LIN {X 0,Y 516.45,Z 515.759,A -85,B 0,C 180,E1 -4943.75,E2 -4943.75} C_VEL
LIN {X 0,Y 516.313,Z 520.47,A -85,B 0,C 180,E1 -4944.924,E2 -4944.924} C_VEL
LIN {X 0,Y 516.373,Z 524.074,A -85,B 0,C 180,E1 -4946.098,E2 -4946.098} C_VEL
LIN {X 0,Y 516.282,Z 525.941,A -85,B 0,C 180,E1 -4946.879,E2 -4946.879} C_VEL
LIN {X 0,Y 516.261,Z 527.348,A -85,B 0,C 180,E1 -4947.659,E2 -4947.659} C_VEL
LIN {X 0,Y 516.16,Z 528.967,A -85,B 0,C 180,E1 -4949.22,E2 -4949.22} C_VEL
LIN {X 0,Y 516.155,Z 529.205,A -85,B 0,C 180,E1 -4950,E2 -4950} C_VEL
LIN {X 0,Y 516.16,Z 529.022,A -85,B 0,C 180,E1 -4950.78,E2 -4950.78} C_VEL
LIN {X 0,Y 516.262,Z 527.473,A -85,B 0,C 180,E1 -4952.341,E2 -4952.341} C_VEL
LIN {X 0,Y 516.283,Z 526.12,A -85,B 0,C 180,E1 -4953.121,E2 -4953.121} C_VEL
LIN {X 0,Y 516.361,Z 523.259,A -85,B 0,C 180,E1 -4954.293,E2 -4954.293} C_VEL
LIN {X 0,Y 516.404,Z 519.379,A -85,B 0,C 180,E1 -4955.467,E2 -4955.467} C_VEL
LIN {X 0,Y 516.485,Z 513.559,A -85,B 0,C 180,E1 -4956.808,E2 -4956.808} C_VEL
LIN {X 0,Y 516.654,Z 506.85,A -85,B 0,C 180,E1 -4958.015,E2 -4958.015} C_VEL
LIN {X 0,Y 516.847,Z 498.704,A -85,B 0,C 180,E1 -4959.194,E2 -4959.194} C_VEL
LIN {X 0,Y 517.103,Z 490.365,A -85,B 0,C 180,E1 -4960.177,E2 -4960.177} C_VEL
LIN {X 0,Y 517.462,Z 480.067,A -85,B 0,C 180,E1 -4961.159,E2 -4961.159} C_VEL
LIN {X 0,Y 517.768,Z 468.543,A -85,B 0,C 180,E1 -4962.039,E2 -4962.039} C_VEL
LIN {X 0,Y 518.054,Z 456.894,A -85,B 0,C 180,E1 -4962.736,E2 -4962.736} C_VEL
LIN {X 0,Y 518.318,Z 444.877,A -85,B 0,C 180,E1 -4963.277,E2 -4963.277} C_VEL
LIN {X 0,Y 518.3,Z 435.908,A -85,B 0,C 180,E1 -4963.59,E2 -4963.59} C_VEL
LIN {X 0,Y 516.365,Z 425.054,A -85,B 0,C 180,E1 -4963.93,E2 -4963.93} C_VEL
LIN {X 0,Y 516.347,Z 420.588,A -85,B 0,C 180,E1 -4966.609,E2 -4966.609} C_VEL
LIN {X 0,Y 516.394,Z 416.475,A -85,B 0,C 180,E1 -4969.065,E2 -4969.065} C_VEL
LIN {X 0,Y 516.487,Z 411.014,A -85,B 0,C 180,E1 -4972.396,E2 -4972.396} C_VEL
LIN {X 0,Y 516.554,Z 406.929,A -85,B 0,C 180,E1 -4974.947,E2 -4974.947} C_VEL
LIN {X 0,Y 516.637,Z 402.398,A -85,B 0,C 180,E1 -4977.844,E2 -4977.844} C_VEL
LIN {X 0,Y 516.679,Z 398.764,A -85,B 0,C 180,E1 -4980.218,E2 -4980.218} C_VEL
LIN {X 0,Y 516.778,Z 394.644,A -85,B 0,C 180,E1 -4982.956,E2 -4982.956} C_VEL
LIN {X 0,Y 516.764,Z 391.166,A -85,B 0,C 180,E1 -4985.313,E2 -4985.313} C_VEL
LIN {X 0,Y 516.883,Z 391.097,A -85,B 0,C 180,E1 -4987.943,E2 -4987.943} C_VEL
LIN {X 0,Y 516.888,Z 391.1,A -85,B 0,C 180,E1 -4990.742,E2 -4990.742} C_VEL
LIN {X 0,Y 516.908,Z 391.096,A -85,B 0,C 180,E1 -4992.829,E2 -4992.829} C_VEL
LIN {X 0,Y 516.885,Z 391.099,A -85,B 0,C 180,E1 -4996.107,E2 -4996.107} C_VEL
LIN {X 0,Y 516.916,Z 391.095,A -85,B 0,C 180,E1 -4998.399,E2 -4998.399} C_VEL
LIN {X 0,Y 516.886,Z 391.097,A -85,B 0,C 180,E1 -5001.284,E2 -5001.284} C_VEL
LIN {X 0,Y 516.874,Z 391.104,A -85,B 0,C 180,E1 -5004.22,E2 -5004.22} C_VEL
LIN {X 0,Y 516.898,Z 391.099,A -85,B 0,C 180,E1 -5007.053,E2 -5007.053} C_VEL
LIN {X 0,Y 516.895,Z 391.098,A -85,B 0,C 180,E1 -5009.796,E2 -5009.796} C_VEL
LIN {X 0,Y 516.932,Z 391.096,A -85,B 0,C 180,E1 -5012.467,E2 -5012.467} C_VEL
LIN {X 0,Y 516.879,Z 391.098,A -85,B 0,C 180,E1 -5015.07,E2 -5015.07} C_VEL
LIN {X 0,Y 516.872,Z 391.102,A -85,B 0,C 180,E1 -5017.622,E2 -5017.622} C_VEL
LIN {X 0,Y 516.936,Z 391.093,A -85,B 0,C 180,E1 -5020.13,E2 -5020.13} C_VEL
LIN {X 0,Y 516.911,Z 391.098,A -85,B 0,C 180,E1 -5022.595,E2 -5022.595} C_VEL
LIN {X 0,Y 516.946,Z 391.092,A -85,B 0,C 180,E1 -5025.03,E2 -5025.03} C_VEL
LIN {X 0,Y 516.969,Z 391.091,A -85,B 0,C 180,E1 -5028.234,E2 -5028.234} C_VEL
LIN {X 0,Y 516.973,Z 391.09,A -85,B 0,C 180,E1 -5031.4,E2 -5031.4} C_VEL
LIN {X 0,Y 517.013,Z 391.083,A -85,B 0,C 180,E1 -5033.757,E2 -5033.757} C_VEL
LIN {X 0,Y 517.085,Z 391.074,A -85,B 0,C 180,E1 -5037.663,E2 -5037.663} C_VEL
LIN {X 0,Y 517.097,Z 391.07,A -85,B 0,C 180,E1 -5040.779,E2 -5040.779} C_VEL
LIN {X 0,Y 517.015,Z 391.083,A -85,B 0,C 180,E1 -5043.117,E2 -5043.117} C_VEL
LIN {X 0,Y 517.013,Z 391.083,A -85,B 0,C 180,E1 -5046.243,E2 -5046.243} C_VEL
LIN {X 0,Y 516.956,Z 391.09,A -85,B 0,C 180,E1 -5049.389,E2 -5049.389} C_VEL
LIN {X 0,Y 516.988,Z 391.089,A -85,B 0,C 180,E1 -5051.824,E2 -5051.824} C_VEL
LIN {X 0,Y 516.948,Z 391.091,A -85,B 0,C 180,E1 -5055.146,E2 -5055.146} C_VEL
LIN {X 0,Y 516.929,Z 391.093,A -85,B 0,C 180,E1 -5058.222,E2 -5058.222} C_VEL
LIN {X 0,Y 516.916,Z 391.098,A -85,B 0,C 180,E1 -5060.701,E2 -5060.701} C_VEL
LIN {X 0,Y 516.894,Z 391.1,A -85,B 0,C 180,E1 -5064.073,E2 -5064.073} C_VEL
LIN {X 0,Y 516.929,Z 391.092,A -85,B 0,C 180,E1 -5066.658,E2 -5066.658} C_VEL
LIN {X 0,Y 516.914,Z 391.096,A -85,B 0,C 180,E1 -5069.524,E2 -5069.524} C_VEL
LIN {X 0,Y 516.899,Z 391.1,A -85,B 0,C 180,E1 -5072.543,E2 -5072.543} C_VEL
LIN {X 0,Y 516.882,Z 391.099,A -85,B 0,C 180,E1 -5075.332,E2 -5075.332} C_VEL
LIN {X 0,Y 516.884,Z 391.101,A -85,B 0,C 180,E1 -5077.943,E2 -5077.943} C_VEL
LIN {X 0,Y 516.888,Z 391.099,A -85,B 0,C 180,E1 -5080.741,E2 -5080.741} C_VEL
LIN {X 0,Y 516.887,Z 391.103,A -85,B 0,C 180,E1 -5082.831,E2 -5082.831} C_VEL
LIN {X 0,Y 516.926,Z 391.094,A -85,B 0,C 180,E1 -5085.01,E2 -5085.01} C_VEL
LIN {X 0,Y 516.919,Z 391.097,A -85,B 0,C 180,E1 -5088.398,E2 -5088.398} C_VEL
LIN {X 0,Y 516.884,Z 391.104,A -85,B 0,C 180,E1 -5091.284,E2 -5091.284} C_VEL
LIN {X 0,Y 516.901,Z 391.162,A -85,B 0,C 180,E1 -5092.4,E2 -5092.4} C_VEL
LIN {X 0,Y 517.556,Z 395.906,A -85,B 0,C 180,E1 -5094.563,E2 -5094.563} C_VEL
LIN {X 0,Y 517.418,Z 402.548,A -85,B 0,C 180,E1 -5097.367,E2 -5097.367} C_VEL
LIN {X 0,Y 517.231,Z 410.058,A -85,B 0,C 180,E1 -5100.414,E2 -5100.414} C_VEL
LIN {X 0,Y 517.02,Z 417.541,A -85,B 0,C 180,E1 -5103.347,E2 -5103.347} C_VEL
LIN {X 0,Y 516.858,Z 425.407,A -85,B 0,C 180,E1 -5106.351,E2 -5106.351} C_VEL
LIN {X 0,Y 516.751,Z 433.272,A -85,B 0,C 180,E1 -5109.292,E2 -5109.292} C_VEL
LIN {X 0,Y 516.585,Z 441.385,A -85,B 0,C 180,E1 -5112.238,E2 -5112.238} C_VEL
LIN {X 0,Y 516.514,Z 449.143,A -85,B 0,C 180,E1 -5115.032,E2 -5115.032} C_VEL
LIN {X 0,Y 516.487,Z 452.291,A -85,B 0,C 180,E1 -5116.111,E2 -5116.111} C_VEL
LIN {X 0,Y 518.462,Z 464.61,A -85,B 0,C 180,E1 -5116.452,E2 -5116.452} C_VEL
LIN {X 0,Y 518.211,Z 477.648,A -85,B 0,C 180,E1 -5116.92,E2 -5116.92} C_VEL
LIN {X 0,Y 517.922,Z 490.006,A -85,B 0,C 180,E1 -5117.532,E2 -5117.532} C_VEL
LIN {X 0,Y 517.653,Z 501.19,A -85,B 0,C 180,E1 -5118.249,E2 -5118.249} C_VEL
LIN {X 0,Y 517.34,Z 512.104,A -85,B 0,C 180,E1 -5119.135,E2 -5119.135} C_VEL
LIN {X 0,Y 517.031,Z 521.003,A -85,B 0,C 180,E1 -5120.02,E2 -5120.02} C_VEL
LIN {X 0,Y 516.773,Z 530.675,A -85,B 0,C 180,E1 -5121.199,E2 -5121.199} C_VEL
LIN {X 0,Y 516.563,Z 538.374,A -85,B 0,C 180,E1 -5122.377,E2 -5122.377} C_VEL
LIN {X 0,Y 516.427,Z 545.472,A -85,B 0,C 180,E1 -5123.75,E2 -5123.75} C_VEL
LIN {X 0,Y 516.313,Z 550.193,A -85,B 0,C 180,E1 -5124.924,E2 -5124.924} C_VEL
LIN {X 0,Y 516.354,Z 553.803,A -85,B 0,C 180,E1 -5126.098,E2 -5126.098} C_VEL
LIN {X 0,Y 516.282,Z 555.663,A -85,B 0,C 180,E1 -5126.879,E2 -5126.879} C_VEL
LIN {X 0,Y 516.261,Z 557.058,A -85,B 0,C 180,E1 -5127.659,E2 -5127.659} C_VEL
LIN {X 0,Y 516.16,Z 558.659,A -85,B 0,C 180,E1 -5129.22,E2 -5129.22} C_VEL
LIN {X 0,Y 516.154,Z 558.875,A -85,B 0,C 180,E1 -5130,E2 -5130} C_VEL
LIN {X 0,Y 516.192,Z 558.054,A -85,B 0,C 180,E1 -5131.56,E2 -5131.56} C_VEL
LIN {X 0,Y 516.261,Z 557.061,A -85,B 0,C 180,E1 -5132.341,E2 -5132.341} C_VEL
LIN {X 0,Y 516.282,Z 555.667,A -85,B 0,C 180,E1 -5133.121,E2 -5133.121} C_VEL
LIN {X 0,Y 516.326,Z 552.733,A -85,B 0,C 180,E1 -5134.293,E2 -5134.293} C_VEL
LIN {X 0,Y 516.383,Z 548.761,A -85,B 0,C 180,E1 -5135.467,E2 -5135.467} C_VEL
LIN {X 0,Y 516.465,Z 543.473,A -85,B 0,C 180,E1 -5136.679,E2 -5136.679} C_VEL
LIN {X 0,Y 516.597,Z 537.214,A -85,B 0,C 180,E1 -5137.819,E2 -5137.819} C_VEL
LIN {X 0,Y 516.807,Z 529.186,A -85,B 0,C 180,E1 -5138.997,E2 -5138.997} C_VEL
LIN {X 0,Y 517.031,Z 521.005,A -85,B 0,C 180,E1 -5139.98,E2 -5139.98} C_VEL
LIN {X 0,Y 517.382,Z 511.032,A -85,B 0,C 180,E1 -5140.963,E2 -5140.963} C_VEL
LIN {X 0,Y 517.647,Z 501.194,A -85,B 0,C 180,E1 -5141.751,E2 -5141.751} C_VEL
LIN {X 0,Y 517.933,Z 490.041,A -85,B 0,C 180,E1 -5142.466,E2 -5142.466} C_VEL
LIN {X 0,Y 518.191,Z 477.642,A -85,B 0,C 180,E1 -5143.081,E2 -5143.081} C_VEL
LIN {X 0,Y 518.495,Z 464.607,A -85,B 0,C 180,E1 -5143.547,E2 -5143.547} C_VEL
LIN {X 0,Y 516.475,Z 452.075,A -85,B 0,C 180,E1 -5143.902,E2 -5143.902} C_VEL
LIN {X 0,Y 516.54,Z 444.494,A -85,B 0,C 180,E1 -5146.602,E2 -5146.602} C_VEL
LIN {X 0,Y 516.686,Z 436.567,A -85,B 0,C 180,E1 -5149.466,E2 -5149.466} C_VEL
LIN {X 0,Y 516.797,Z 428.777,A -85,B 0,C 180,E1 -5152.382,E2 -5152.382} C_VEL
LIN {X 0,Y 516.958,Z 420.911,A -85,B 0,C 180,E1 -5155.356,E2 -5155.356} C_VEL
LIN {X 0,Y 517.163,Z 413.048,A -85,B 0,C 180,E1 -5158.401,E2 -5158.401} C_VEL
LIN {X 0,Y 517.356,Z 405.213,A -85,B 0,C 180,E1 -5161.533,E2 -5161.533} C_VEL
LIN {X 0,Y 517.492,Z 399.121,A -85,B 0,C 180,E1 -5164.062,E2 -5164.062} C_VEL
LIN {X 0,Y 517.531,Z 395.238,A -85,B 0,C 180,E1 -5165.728,E2 -5165.728} C_VEL
LIN {X 0,Y 516.884,Z 391.103,A -85,B 0,C 180,E1 -5167.662,E2 -5167.662} C_VEL
LIN {X 0,Y 516.886,Z 391.1,A -85,B 0,C 180,E1 -5170.741,E2 -5170.741} C_VEL
LIN {X 0,Y 516.907,Z 391.096,A -85,B 0,C 180,E1 -5172.829,E2 -5172.829} C_VEL
LIN {X 0,Y 516.925,Z 391.095,A -85,B 0,C 180,E1 -5175.01,E2 -5175.01} C_VEL
LIN {X 0,Y 516.917,Z 391.094,A -85,B 0,C 180,E1 -5178.398,E2 -5178.398} C_VEL
LIN {X 0,Y 516.884,Z 391.098,A -85,B 0,C 180,E1 -5181.284,E2 -5181.284} C_VEL
LIN {X 0,Y 516.891,Z 391.101,A -85,B 0,C 180,E1 -5184.221,E2 -5184.221} C_VEL
LIN {X 0,Y 516.897,Z 391.099,A -85,B 0,C 180,E1 -5187.053,E2 -5187.053} C_VEL
LIN {X 0,Y 516.894,Z 391.096,A -85,B 0,C 180,E1 -5189.796,E2 -5189.796} C_VEL
LIN {X 0,Y 516.93,Z 391.096,A -85,B 0,C 180,E1 -5192.467,E2 -5192.467} C_VEL
LIN {X 0,Y 516.877,Z 391.099,A -85,B 0,C 180,E1 -5195.07,E2 -5195.07} C_VEL
LIN {X 0,Y 516.87,Z 391.103,A -85,B 0,C 180,E1 -5197.622,E2 -5197.622} C_VEL
LIN {X 0,Y 516.935,Z 391.092,A -85,B 0,C 180,E1 -5200.13,E2 -5200.13} C_VEL
LIN {X 0,Y 516.932,Z 391.095,A -85,B 0,C 180,E1 -5202.596,E2 -5202.596} C_VEL
LIN {X 0,Y 516.945,Z 391.091,A -85,B 0,C 180,E1 -5205.03,E2 -5205.03} C_VEL
LIN {X 0,Y 517.007,Z 391.087,A -85,B 0,C 180,E1 -5208.235,E2 -5208.235} C_VEL
LIN {X 0,Y 516.972,Z 391.09,A -85,B 0,C 180,E1 -5211.4,E2 -5211.4} C_VEL
LIN {X 0,Y 517.012,Z 391.083,A -85,B 0,C 180,E1 -5213.757,E2 -5213.757} C_VEL
LIN {X 0,Y 517.085,Z 391.072,A -85,B 0,C 180,E1 -5217.663,E2 -5217.663} C_VEL
LIN {X 0,Y 517.096,Z 391.071,A -85,B 0,C 180,E1 -5220.779,E2 -5220.779} C_VEL
LIN {X 0,Y 517.014,Z 391.085,A -85,B 0,C 180,E1 -5223.117,E2 -5223.117} C_VEL
LIN {X 0,Y 517.012,Z 391.083,A -85,B 0,C 180,E1 -5226.243,E2 -5226.243} C_VEL
LIN {X 0,Y 516.956,Z 391.089,A -85,B 0,C 180,E1 -5229.389,E2 -5229.389} C_VEL
LIN {X 0,Y 516.986,Z 391.089,A -85,B 0,C 180,E1 -5231.824,E2 -5231.824} C_VEL
LIN {X 0,Y 516.947,Z 391.092,A -85,B 0,C 180,E1 -5235.147,E2 -5235.147} C_VEL
LIN {X 0,Y 516.919,Z 391.095,A -85,B 0,C 180,E1 -5238.223,E2 -5238.223} C_VEL
LIN {X 0,Y 516.915,Z 391.097,A -85,B 0,C 180,E1 -5240.701,E2 -5240.701} C_VEL
LIN {X 0,Y 516.893,Z 391.101,A -85,B 0,C 180,E1 -5244.073,E2 -5244.073} C_VEL
LIN {X 0,Y 516.928,Z 391.091,A -85,B 0,C 180,E1 -5246.658,E2 -5246.658} C_VEL
LIN {X 0,Y 516.913,Z 391.097,A -85,B 0,C 180,E1 -5249.524,E2 -5249.524} C_VEL
LIN {X 0,Y 516.898,Z 391.1,A -85,B 0,C 180,E1 -5252.543,E2 -5252.543} C_VEL
LIN {X 0,Y 516.886,Z 391.098,A -85,B 0,C 180,E1 -5255.333,E2 -5255.333} C_VEL
LIN {X 0,Y 516.884,Z 391.1,A -85,B 0,C 180,E1 -5257.943,E2 -5257.943} C_VEL
LIN {X 0,Y 516.887,Z 391.098,A -85,B 0,C 180,E1 -5260.742,E2 -5260.742} C_VEL
LIN {X 0,Y 516.885,Z 391.102,A -85,B 0,C 180,E1 -5262.832,E2 -5262.832} C_VEL
LIN {X 0,Y 516.925,Z 391.095,A -85,B 0,C 180,E1 -5265.01,E2 -5265.01} C_VEL
LIN {X 0,Y 516.918,Z 391.096,A -85,B 0,C 180,E1 -5268.399,E2 -5268.399} C_VEL
LIN {X 0,Y 516.884,Z 391.098,A -85,B 0,C 180,E1 -5270.301,E2 -5270.301} C_VEL
LIN {X 0,Y 516.213,Z 391.184,A -85,B 0,C 180,E1 -5270.951,E2 -5270.951} C_VEL
LIN {X 0,Y 513.364,Z 391.538,A -85,B 0,C 180,E1 -5272.007,E2 -5272.007} C_VEL
LIN {X 0,Y 510.941,Z 391.842,A -85,B 0,C 180,E1 -5272.857,E2 -5272.857} C_VEL
LIN {X 0,Y 509.874,Z 391.975,A -85,B 0,C 180,E1 -5273.513,E2 -5273.513} C_VEL
LIN {X 0,Y 509.774,Z 391.985,A -85,B 0,C 180,E1 -5273.736,E2 -5273.736} C_VEL
LIN {X 0,Y 509.742,Z 391.992,A -85,B 0,C 180,E1 -5274.615,E2 -5274.615} C_VEL
LIN {X 0,Y 509.714,Z 395.641,A -85,B 0,C 180,E1 -5277.254,E2 -5277.254} C_VEL
LIN {X 0,Y 509.61,Z 400.227,A -85,B 0,C 180,E1 -5280.323,E2 -5280.323} C_VEL
LIN {X 0,Y 509.541,Z 404.185,A -85,B 0,C 180,E1 -5282.925,E2 -5282.925} C_VEL
LIN {X 0,Y 509.502,Z 408.276,A -85,B 0,C 180,E1 -5285.561,E2 -5285.561} C_VEL
LIN {X 0,Y 509.373,Z 412.339,A -85,B 0,C 180,E1 -5288.128,E2 -5288.128} C_VEL
LIN {X 0,Y 509.324,Z 416.434,A -85,B 0,C 180,E1 -5290.66,E2 -5290.66} C_VEL
LIN {X 0,Y 509.306,Z 420.558,A -85,B 0,C 180,E1 -5293.155,E2 -5293.155} C_VEL
LIN {X 0,Y 509.279,Z 425.464,A -85,B 0,C 180,E1 -5295.987,E2 -5295.987} C_VEL
LIN {X 0,Y 511.505,Z 437.605,A -85,B 0,C 180,E1 -5296.366,E2 -5296.366} C_VEL
LIN {X 0,Y 511.345,Z 450.083,A -85,B 0,C 180,E1 -5296.842,E2 -5296.842} C_VEL
LIN {X 0,Y 511.029,Z 462.423,A -85,B 0,C 180,E1 -5297.48,E2 -5297.48} C_VEL
LIN {X 0,Y 510.715,Z 474.284,A -85,B 0,C 180,E1 -5298.289,E2 -5298.289} C_VEL
LIN {X 0,Y 510.319,Z 484.759,A -85,B 0,C 180,E1 -5299.185,E2 -5299.185} C_VEL
LIN {X 0,Y 510.061,Z 493.315,A -85,B 0,C 180,E1 -5300.082,E2 -5300.082} C_VEL
LIN {X 0,Y 509.82,Z 501.194,A -85,B 0,C 180,E1 -5301.078,E2 -5301.078} C_VEL
LIN {X 0,Y 509.56,Z 508.9,A -85,B 0,C 180,E1 -5302.272,E2 -5302.272} C_VEL
LIN {X 0,Y 509.387,Z 515.966,A -85,B 0,C 180,E1 -5303.663,E2 -5303.663} C_VEL
LIN {X 0,Y 509.248,Z 520.676,A -85,B 0,C 180,E1 -5304.853,E2 -5304.853} C_VEL
LIN {X 0,Y 509.303,Z 524.279,A -85,B 0,C 180,E1 -5306.044,E2 -5306.044} C_VEL
LIN {X 0,Y 509.201,Z 526.146,A -85,B 0,C 180,E1 -5306.835,E2 -5306.835} C_VEL
LIN {X 0,Y 509.19,Z 527.552,A -85,B 0,C 180,E1 -5307.627,E2 -5307.627} C_VEL
LIN {X 0,Y 509.074,Z 529.171,A -85,B 0,C 180,E1 -5309.209,E2 -5309.209} C_VEL
LIN {X 0,Y 509.066,Z 529.408,A -85,B 0,C 180,E1 -5310,E2 -5310} C_VEL
LIN {X 0,Y 509.074,Z 529.225,A -85,B 0,C 180,E1 -5310.791,E2 -5310.791} C_VEL
LIN {X 0,Y 509.19,Z 527.676,A -85,B 0,C 180,E1 -5312.373,E2 -5312.373} C_VEL
LIN {X 0,Y 509.202,Z 526.323,A -85,B 0,C 180,E1 -5313.165,E2 -5313.165} C_VEL
LIN {X 0,Y 509.282,Z 523.461,A -85,B 0,C 180,E1 -5314.353,E2 -5314.353} C_VEL
LIN {X 0,Y 509.346,Z 519.581,A -85,B 0,C 180,E1 -5315.543,E2 -5315.543} C_VEL
LIN {X 0,Y 509.412,Z 514.576,A -85,B 0,C 180,E1 -5316.734,E2 -5316.734} C_VEL
LIN {X 0,Y 509.597,Z 508.273,A -85,B 0,C 180,E1 -5317.927,E2 -5317.927} C_VEL
LIN {X 0,Y 509.777,Z 500.383,A -85,B 0,C 180,E1 -5319.122,E2 -5319.122} C_VEL
LIN {X 0,Y 510.085,Z 492.336,A -85,B 0,C 180,E1 -5320.118,E2 -5320.118} C_VEL
LIN {X 0,Y 510.414,Z 482.517,A -85,B 0,C 180,E1 -5321.115,E2 -5321.115} C_VEL
LIN {X 0,Y 510.706,Z 472.858,A -85,B 0,C 180,E1 -5321.913,E2 -5321.913} C_VEL
LIN {X 0,Y 511.034,Z 461.886,A -85,B 0,C 180,E1 -5322.641,E2 -5322.641} C_VEL
LIN {X 0,Y 511.332,Z 449.841,A -85,B 0,C 180,E1 -5323.26,E2 -5323.26} C_VEL
LIN {X 0,Y 511.473,Z 437.271,A -85,B 0,C 180,E1 -5323.737,E2 -5323.737} C_VEL
LIN {X 0,Y 509.275,Z 425.263,A -85,B 0,C 180,E1 -5324.128,E2 -5324.128} C_VEL
LIN {X 0,Y 509.288,Z 420.721,A -85,B 0,C 180,E1 -5326.846,E2 -5326.846} C_VEL
LIN {X 0,Y 509.318,Z 416.596,A -85,B 0,C 180,E1 -5329.34,E2 -5329.34} C_VEL
LIN {X 0,Y 509.425,Z 411.586,A -85,B 0,C 180,E1 -5332.432,E2 -5332.432} C_VEL
LIN {X 0,Y 509.493,Z 407.051,A -85,B 0,C 180,E1 -5335.317,E2 -5335.317} C_VEL
LIN {X 0,Y 509.572,Z 402.861,A -85,B 0,C 180,E1 -5338.031,E2 -5338.031} C_VEL
LIN {X 0,Y 509.653,Z 398.017,A -85,B 0,C 180,E1 -5341.244,E2 -5341.244} C_VEL
LIN {X 0,Y 509.748,Z 394.722,A -85,B 0,C 180,E1 -5343.469,E2 -5343.469} C_VEL
LIN {X 0,Y 509.738,Z 391.993,A -85,B 0,C 180,E1 -5345.386,E2 -5345.386} C_VEL
LIN {X 0,Y 509.853,Z 391.976,A -85,B 0,C 180,E1 -5348.338,E2 -5348.338} C_VEL
LIN {X 0,Y 509.861,Z 391.974,A -85,B 0,C 180,E1 -5351.425,E2 -5351.425} C_VEL
LIN {X 0,Y 509.842,Z 391.976,A -85,B 0,C 180,E1 -5354.67,E2 -5354.67} C_VEL
LIN {X 0,Y 509.859,Z 391.973,A -85,B 0,C 180,E1 -5358.103,E2 -5358.103} C_VEL
LIN {X 0,Y 509.851,Z 391.98,A -85,B 0,C 180,E1 -5360.648,E2 -5360.648} C_VEL
LIN {X 0,Y 509.828,Z 391.978,A -85,B 0,C 180,E1 -5363.647,E2 -5363.647} C_VEL
LIN {X 0,Y 509.862,Z 391.974,A -85,B 0,C 180,E1 -5366.539,E2 -5366.539} C_VEL
LIN {X 0,Y 509.849,Z 391.977,A -85,B 0,C 180,E1 -5369.334,E2 -5369.334} C_VEL
LIN {X 0,Y 509.897,Z 391.969,A -85,B 0,C 180,E1 -5372.055,E2 -5372.055} C_VEL
LIN {X 0,Y 509.844,Z 391.976,A -85,B 0,C 180,E1 -5374.702,E2 -5374.702} C_VEL
LIN {X 0,Y 509.83,Z 391.979,A -85,B 0,C 180,E1 -5377.458,E2 -5377.458} C_VEL
LIN {X 0,Y 509.921,Z 391.969,A -85,B 0,C 180,E1 -5379.845,E2 -5379.845} C_VEL
LIN {X 0,Y 509.878,Z 391.973,A -85,B 0,C 180,E1 -5383.174,E2 -5383.174} C_VEL
LIN {X 0,Y 509.868,Z 391.972,A -85,B 0,C 180,E1 -5385.634,E2 -5385.634} C_VEL
LIN {X 0,Y 509.916,Z 391.965,A -85,B 0,C 180,E1 -5388.875,E2 -5388.875} C_VEL
LIN {X 0,Y 509.956,Z 391.962,A -85,B 0,C 180,E1 -5392.078,E2 -5392.078} C_VEL
LIN {X 0,Y 509.985,Z 391.96,A -85,B 0,C 180,E1 -5394.464,E2 -5394.464} C_VEL
LIN {X 0,Y 510.056,Z 391.949,A -85,B 0,C 180,E1 -5397.631,E2 -5397.631} C_VEL
LIN {X 0,Y 510.067,Z 391.946,A -85,B 0,C 180,E1 -5400.789,E2 -5400.789} C_VEL
LIN {X 0,Y 509.957,Z 391.962,A -85,B 0,C 180,E1 -5403.16,E2 -5403.16} C_VEL
LIN {X 0,Y 509.981,Z 391.959,A -85,B 0,C 180,E1 -5406.33,E2 -5406.33} C_VEL
LIN {X 0,Y 509.92,Z 391.969,A -85,B 0,C 180,E1 -5408.72,E2 -5408.72} C_VEL
LIN {X 0,Y 509.955,Z 391.966,A -85,B 0,C 180,E1 -5411.93,E2 -5411.93} C_VEL
LIN {X 0,Y 509.897,Z 391.971,A -85,B 0,C 180,E1 -5415.242,E2 -5415.242} C_VEL
LIN {X 0,Y 509.892,Z 391.969,A -85,B 0,C 180,E1 -5418.001,E2 -5418.001} C_VEL
LIN {X 0,Y 509.854,Z 391.976,A -85,B 0,C 180,E1 -5421.002,E2 -5421.002} C_VEL
LIN {X 0,Y 509.826,Z 391.98,A -85,B 0,C 180,E1 -5423.564,E2 -5423.564} C_VEL
LIN {X 0,Y 509.915,Z 391.966,A -85,B 0,C 180,E1 -5426.379,E2 -5426.379} C_VEL
LIN {X 0,Y 509.88,Z 391.972,A -85,B 0,C 180,E1 -5428.844,E2 -5428.844} C_VEL
LIN {X 0,Y 509.823,Z 391.978,A -85,B 0,C 180,E1 -5431.59,E2 -5431.59} C_VEL
LIN {X 0,Y 509.855,Z 391.977,A -85,B 0,C 180,E1 -5434.413,E2 -5434.413} C_VEL
LIN {X 0,Y 509.822,Z 391.981,A -85,B 0,C 180,E1 -5437.341,E2 -5437.341} C_VEL
LIN {X 0,Y 509.841,Z 391.975,A -85,B 0,C 180,E1 -5440.382,E2 -5440.382} C_VEL
LIN {X 0,Y 509.827,Z 391.98,A -85,B 0,C 180,E1 -5443.062,E2 -5443.062} C_VEL
LIN {X 0,Y 509.834,Z 391.978,A -85,B 0,C 180,E1 -5445.792,E2 -5445.792} C_VEL
LIN {X 0,Y 509.86,Z 391.976,A -85,B 0,C 180,E1 -5448.575,E2 -5448.575} C_VEL
LIN {X 0,Y 509.857,Z 391.977,A -85,B 0,C 180,E1 -5451.786,E2 -5451.786} C_VEL
LIN {X 0,Y 509.885,Z 392.202,A -85,B 0,C 180,E1 -5452.291,E2 -5452.291} C_VEL
LIN {X 0,Y 510.552,Z 396.544,A -85,B 0,C 180,E1 -5454.308,E2 -5454.308} C_VEL
LIN {X 0,Y 510.418,Z 403.106,A -85,B 0,C 180,E1 -5457.131,E2 -5457.131} C_VEL
LIN {X 0,Y 510.25,Z 409.598,A -85,B 0,C 180,E1 -5459.819,E2 -5459.819} C_VEL
LIN {X 0,Y 509.982,Z 417.433,A -85,B 0,C 180,E1 -5462.95,E2 -5462.95} C_VEL
LIN {X 0,Y 509.839,Z 424.175,A -85,B 0,C 180,E1 -5465.572,E2 -5465.572} C_VEL
LIN {X 0,Y 509.7,Z 432.031,A -85,B 0,C 180,E1 -5468.568,E2 -5468.568} C_VEL
LIN {X 0,Y 509.573,Z 439.949,A -85,B 0,C 180,E1 -5471.505,E2 -5471.505} C_VEL
LIN {X 0,Y 509.445,Z 449.296,A -85,B 0,C 180,E1 -5474.946,E2 -5474.946} C_VEL
LIN {X 0,Y 509.401,Z 452.081,A -85,B 0,C 180,E1 -5475.914,E2 -5475.914} C_VEL
LIN {X 0,Y 511.546,Z 465.241,A -85,B 0,C 180,E1 -5476.291,E2 -5476.291} C_VEL
LIN {X 0,Y 511.259,Z 478.575,A -85,B 0,C 180,E1 -5476.789,E2 -5476.789} C_VEL
LIN {X 0,Y 510.946,Z 491.12,A -85,B 0,C 180,E1 -5477.434,E2 -5477.434} C_VEL
LIN {X 0,Y 510.618,Z 502.299,A -85,B 0,C 180,E1 -5478.186,E2 -5478.186} C_VEL
LIN {X 0,Y 510.309,Z 512.972,A -85,B 0,C 180,E1 -5479.084,E2 -5479.084} C_VEL
LIN {X 0,Y 509.954,Z 522.587,A -85,B 0,C 180,E1 -5480.08,E2 -5480.08} C_VEL
LIN {X 0,Y 509.711,Z 530.47,A -85,B 0,C 180,E1 -5481.076,E2 -5481.076} C_VEL
LIN {X 0,Y 509.513,Z 538.17,A -85,B 0,C 180,E1 -5482.271,E2 -5482.271} C_VEL
LIN {X 0,Y 509.328,Z 545.267,A -85,B 0,C 180,E1 -5483.662,E2 -5483.662} C_VEL
LIN {X 0,Y 509.245,Z 549.989,A -85,B 0,C 180,E1 -5484.853,E2 -5484.853} C_VEL
LIN {X 0,Y 509.25,Z 553.599,A -85,B 0,C 180,E1 -5486.043,E2 -5486.043} C_VEL
LIN {X 0,Y 509.2,Z 555.459,A -85,B 0,C 180,E1 -5486.835,E2 -5486.835} C_VEL
LIN {X 0,Y 509.19,Z 556.854,A -85,B 0,C 180,E1 -5487.627,E2 -5487.627} C_VEL
LIN {X 0,Y 509.073,Z 558.455,A -85,B 0,C 180,E1 -5489.209,E2 -5489.209} C_VEL
LIN {X 0,Y 509.065,Z 558.671,A -85,B 0,C 180,E1 -5490,E2 -5490} C_VEL
LIN {X 0,Y 509.113,Z 557.85,A -85,B 0,C 180,E1 -5491.582,E2 -5491.582} C_VEL
LIN {X 0,Y 509.19,Z 556.858,A -85,B 0,C 180,E1 -5492.373,E2 -5492.373} C_VEL
LIN {X 0,Y 509.2,Z 555.463,A -85,B 0,C 180,E1 -5493.165,E2 -5493.165} C_VEL
LIN {X 0,Y 509.216,Z 552.528,A -85,B 0,C 180,E1 -5494.353,E2 -5494.353} C_VEL
LIN {X 0,Y 509.305,Z 548.557,A -85,B 0,C 180,E1 -5495.543,E2 -5495.543} C_VEL
LIN {X 0,Y 509.402,Z 542.902,A -85,B 0,C 180,E1 -5496.844,E2 -5496.844} C_VEL
LIN {X 0,Y 509.573,Z 535.772,A -85,B 0,C 180,E1 -5498.127,E2 -5498.127} C_VEL
LIN {X 0,Y 509.793,Z 527.489,A -85,B 0,C 180,E1 -5499.322,E2 -5499.322} C_VEL
LIN {X 0,Y 510.055,Z 519,A -85,B 0,C 180,E1 -5500.319,E2 -5500.319} C_VEL
LIN {X 0,Y 510.423,Z 508.512,A -85,B 0,C 180,E1 -5501.315,E2 -5501.315} C_VEL
LIN {X 0,Y 510.696,Z 497.21,A -85,B 0,C 180,E1 -5502.179,E2 -5502.179} C_VEL
LIN {X 0,Y 511.071,Z 486.762,A -85,B 0,C 180,E1 -5502.811,E2 -5502.811} C_VEL
LIN {X 0,Y 511.313,Z 475.096,A -85,B 0,C 180,E1 -5503.361,E2 -5503.361} C_VEL
LIN {X 0,Y 511.434,Z 464.398,A -85,B 0,C 180,E1 -5503.737,E2 -5503.737} C_VEL
LIN {X 0,Y 509.387,Z 451.894,A -85,B 0,C 180,E1 -5504.099,E2 -5504.099} C_VEL
LIN {X 0,Y 509.468,Z 444.335,A -85,B 0,C 180,E1 -5506.839,E2 -5506.839} C_VEL
LIN {X 0,Y 509.627,Z 436.478,A -85,B 0,C 180,E1 -5509.747,E2 -5509.747} C_VEL
LIN {X 0,Y 509.753,Z 429.156,A -85,B 0,C 180,E1 -5512.521,E2 -5512.521} C_VEL
LIN {X 0,Y 509.942,Z 420.8,A -85,B 0,C 180,E1 -5515.73,E2 -5515.73} C_VEL
LIN {X 0,Y 510.14,Z 412.946,A -85,B 0,C 180,E1 -5518.828,E2 -5518.828} C_VEL
LIN {X 0,Y 510.352,Z 405.128,A -85,B 0,C 180,E1 -5522.018,E2 -5522.018} C_VEL
LIN {X 0,Y 510.568,Z 398.479,A -85,B 0,C 180,E1 -5524.837,E2 -5524.837} C_VEL
LIN {X 0,Y 510.38,Z 395.183,A -85,B 0,C 180,E1 -5526.307,E2 -5526.307} C_VEL
LIN {X 0,Y 509.847,Z 391.98,A -85,B 0,C 180,E1 -5527.837,E2 -5527.837} C_VEL
LIN {X 0,Y 509.841,Z 391.978,A -85,B 0,C 180,E1 -5530.698,E2 -5530.698} C_VEL
LIN {X 0,Y 509.829,Z 391.982,A -85,B 0,C 180,E1 -5533.571,E2 -5533.571} C_VEL
LIN {X 0,Y 509.82,Z 391.977,A -85,B 0,C 180,E1 -5536.428,E2 -5536.428} C_VEL
LIN {X 0,Y 509.841,Z 391.976,A -85,B 0,C 180,E1 -5539.302,E2 -5539.302} C_VEL
LIN {X 0,Y 509.854,Z 391.975,A -85,B 0,C 180,E1 -5541.786,E2 -5541.786} C_VEL
LIN {X 0,Y 509.846,Z 391.976,A -85,B 0,C 180,E1 -5544.623,E2 -5544.623} C_VEL
LIN {X 0,Y 509.863,Z 391.976,A -85,B 0,C 180,E1 -5547.481,E2 -5547.481} C_VEL
LIN {X 0,Y 509.86,Z 391.973,A -85,B 0,C 180,E1 -5550.274,E2 -5550.274} C_VEL
LIN {X 0,Y 509.887,Z 391.971,A -85,B 0,C 180,E1 -5552.944,E2 -5552.944} C_VEL
LIN {X 0,Y 509.853,Z 391.976,A -85,B 0,C 180,E1 -5555.573,E2 -5555.573} C_VEL
LIN {X 0,Y 509.824,Z 391.98,A -85,B 0,C 180,E1 -5558.149,E2 -5558.149} C_VEL
LIN {X 0,Y 509.867,Z 391.974,A -85,B 0,C 180,E1 -5560.682,E2 -5560.682} C_VEL
LIN {X 0,Y 509.887,Z 391.971,A -85,B 0,C 180,E1 -5563.175,E2 -5563.175} C_VEL
LIN {X 0,Y 509.867,Z 391.971,A -85,B 0,C 180,E1 -5565.634,E2 -5565.634} C_VEL
LIN {X 0,Y 509.924,Z 391.965,A -85,B 0,C 180,E1 -5568.875,E2 -5568.875} C_VEL
LIN {X 0,Y 509.954,Z 391.962,A -85,B 0,C 180,E1 -5572.079,E2 -5572.079} C_VEL
LIN {X 0,Y 509.984,Z 391.96,A -85,B 0,C 180,E1 -5574.464,E2 -5574.464} C_VEL
LIN {X 0,Y 510.056,Z 391.948,A -85,B 0,C 180,E1 -5577.631,E2 -5577.631} C_VEL
LIN {X 0,Y 510.066,Z 391.947,A -85,B 0,C 180,E1 -5580.79,E2 -5580.79} C_VEL
LIN {X 0,Y 509.956,Z 391.964,A -85,B 0,C 180,E1 -5583.16,E2 -5583.16} C_VEL
LIN {X 0,Y 509.981,Z 391.96,A -85,B 0,C 180,E1 -5586.33,E2 -5586.33} C_VEL
LIN {X 0,Y 509.919,Z 391.968,A -85,B 0,C 180,E1 -5588.72,E2 -5588.72} C_VEL
LIN {X 0,Y 509.954,Z 391.966,A -85,B 0,C 180,E1 -5591.931,E2 -5591.931} C_VEL
LIN {X 0,Y 509.896,Z 391.971,A -85,B 0,C 180,E1 -5595.242,E2 -5595.242} C_VEL
LIN {X 0,Y 509.869,Z 391.973,A -85,B 0,C 180,E1 -5597.993,E2 -5597.993} C_VEL
LIN {X 0,Y 509.889,Z 391.974,A -85,B 0,C 180,E1 -5600.402,E2 -5600.402} C_VEL
LIN {X 0,Y 509.825,Z 391.979,A -85,B 0,C 180,E1 -5603.564,E2 -5603.564} C_VEL
LIN {X 0,Y 509.914,Z 391.965,A -85,B 0,C 180,E1 -5606.379,E2 -5606.379} C_VEL
LIN {X 0,Y 509.879,Z 391.972,A -85,B 0,C 180,E1 -5608.844,E2 -5608.844} C_VEL
LIN {X 0,Y 509.822,Z 391.979,A -85,B 0,C 180,E1 -5611.59,E2 -5611.59} C_VEL
LIN {X 0,Y 509.856,Z 391.976,A -85,B 0,C 180,E1 -5614.413,E2 -5614.413} C_VEL
LIN {X 0,Y 509.822,Z 391.98,A -85,B 0,C 180,E1 -5617.341,E2 -5617.341} C_VEL
LIN {X 0,Y 509.841,Z 391.974,A -85,B 0,C 180,E1 -5620.382,E2 -5620.382} C_VEL
LIN {X 0,Y 509.825,Z 391.982,A -85,B 0,C 180,E1 -5623.062,E2 -5623.062} C_VEL
LIN {X 0,Y 509.833,Z 391.978,A -85,B 0,C 180,E1 -5625.792,E2 -5625.792} C_VEL
LIN {X 0,Y 509.86,Z 391.974,A -85,B 0,C 180,E1 -5628.575,E2 -5628.575} C_VEL
LIN {X 0,Y 509.853,Z 391.976,A -85,B 0,C 180,E1 -5631.787,E2 -5631.787} C_VEL
LIN {X 0,Y 509.774,Z 391.985,A -85,B 0,C 180,E1 -5633.736,E2 -5633.736} C_VEL
LIN {X 0,Y 509.072,Z 392.255,A -85,B 0,C 180,E1 -5634.394,E2 -5634.394} C_VEL
LIN {X 0,Y 506.224,Z 393.55,A -85,B 0,C 180,E1 -5635.456,E2 -5635.456} C_VEL
LIN {X 0,Y 503.821,Z 394.979,A -85,B 0,C 180,E1 -5636.307,E2 -5636.307} C_VEL
LIN {X 0,Y 502.772,Z 396.062,A -85,B 0,C 180,E1 -5636.964,E2 -5636.964} C_VEL
LIN {X 0,Y 502.675,Z 396.395,A -85,B 0,C 180,E1 -5637.187,E2 -5637.187} C_VEL
LIN {X 0,Y 502.567,Z 400.698,A -85,B 0,C 180,E1 -5640.115,E2 -5640.115} C_VEL
LIN {X 0,Y 502.489,Z 404.3,A -85,B 0,C 180,E1 -5642.513,E2 -5642.513} C_VEL
LIN {X 0,Y 502.427,Z 408.712,A -85,B 0,C 180,E1 -5645.399,E2 -5645.399} C_VEL
LIN {X 0,Y 502.351,Z 412.465,A -85,B 0,C 180,E1 -5647.807,E2 -5647.807} C_VEL
LIN {X 0,Y 502.265,Z 416.565,A -85,B 0,C 180,E1 -5650.377,E2 -5650.377} C_VEL
LIN {X 0,Y 502.244,Z 420.704,A -85,B 0,C 180,E1 -5652.911,E2 -5652.911} C_VEL
LIN {X 0,Y 502.249,Z 425.704,A -85,B 0,C 180,E1 -5655.787,E2 -5655.787} C_VEL
LIN {X 0,Y 504.606,Z 438.588,A -85,B 0,C 180,E1 -5656.201,E2 -5656.201} C_VEL
LIN {X 0,Y 504.413,Z 451.428,A -85,B 0,C 180,E1 -5656.709,E2 -5656.709} C_VEL
LIN {X 0,Y 504.102,Z 463.192,A -85,B 0,C 180,E1 -5657.339,E2 -5657.339} C_VEL
LIN {X 0,Y 503.771,Z 474.496,A -85,B 0,C 180,E1 -5658.125,E2 -5658.125} C_VEL
LIN {X 0,Y 503.352,Z 484.97,A -85,B 0,C 180,E1 -5659.033,E2 -5659.033} C_VEL
LIN {X 0,Y 503.071,Z 493.524,A -85,B 0,C 180,E1 -5659.943,E2 -5659.943} C_VEL
LIN {X 0,Y 502.803,Z 501.403,A -85,B 0,C 180,E1 -5660.953,E2 -5660.953} C_VEL
LIN {X 0,Y 502.52,Z 509.108,A -85,B 0,C 180,E1 -5662.163,E2 -5662.163} C_VEL
LIN {X 0,Y 502.324,Z 516.173,A -85,B 0,C 180,E1 -5663.574,E2 -5663.574} C_VEL
LIN {X 0,Y 502.186,Z 520.882,A -85,B 0,C 180,E1 -5664.781,E2 -5664.781} C_VEL
LIN {X 0,Y 502.235,Z 524.485,A -85,B 0,C 180,E1 -5665.988,E2 -5665.988} C_VEL
LIN {X 0,Y 502.124,Z 526.351,A -85,B 0,C 180,E1 -5666.791,E2 -5666.791} C_VEL
LIN {X 0,Y 502.121,Z 527.757,A -85,B 0,C 180,E1 -5667.594,E2 -5667.594} C_VEL
LIN {X 0,Y 501.991,Z 529.375,A -85,B 0,C 180,E1 -5669.198,E2 -5669.198} C_VEL
LIN {X 0,Y 501.98,Z 529.612,A -85,B 0,C 180,E1 -5670,E2 -5670} C_VEL
LIN {X 0,Y 501.99,Z 529.428,A -85,B 0,C 180,E1 -5670.802,E2 -5670.802} C_VEL
LIN {X 0,Y 502.121,Z 527.878,A -85,B 0,C 180,E1 -5672.407,E2 -5672.407} C_VEL
LIN {X 0,Y 502.125,Z 526.526,A -85,B 0,C 180,E1 -5673.21,E2 -5673.21} C_VEL
LIN {X 0,Y 502.206,Z 523.663,A -85,B 0,C 180,E1 -5674.414,E2 -5674.414} C_VEL
LIN {X 0,Y 502.289,Z 519.782,A -85,B 0,C 180,E1 -5675.621,E2 -5675.621} C_VEL
LIN {X 0,Y 502.354,Z 514.778,A -85,B 0,C 180,E1 -5676.829,E2 -5676.829} C_VEL
LIN {X 0,Y 502.556,Z 508.473,A -85,B 0,C 180,E1 -5678.039,E2 -5678.039} C_VEL
LIN {X 0,Y 502.759,Z 500.582,A -85,B 0,C 180,E1 -5679.251,E2 -5679.251} C_VEL
LIN {X 0,Y 503.067,Z 492.535,A -85,B 0,C 180,E1 -5680.26,E2 -5680.26} C_VEL
LIN {X 0,Y 503.453,Z 482.714,A -85,B 0,C 180,E1 -5681.27,E2 -5681.27} C_VEL
LIN {X 0,Y 503.807,Z 471.68,A -85,B 0,C 180,E1 -5682.18,E2 -5682.18} C_VEL
LIN {X 0,Y 504.151,Z 460.853,A -85,B 0,C 180,E1 -5682.888,E2 -5682.888} C_VEL
LIN {X 0,Y 504.471,Z 448.903,A -85,B 0,C 180,E1 -5683.495,E2 -5683.495} C_VEL
LIN {X 0,Y 504.516,Z 437.838,A -85,B 0,C 180,E1 -5683.917,E2 -5683.917} C_VEL
LIN {X 0,Y 502.213,Z 425.471,A -85,B 0,C 180,E1 -5684.331,E2 -5684.331} C_VEL
LIN {X 0,Y 502.261,Z 419.513,A -85,B 0,C 180,E1 -5687.916,E2 -5687.916} C_VEL
LIN {X 0,Y 502.273,Z 415.327,A -85,B 0,C 180,E1 -5690.476,E2 -5690.476} C_VEL
LIN {X 0,Y 502.364,Z 411.25,A -85,B 0,C 180,E1 -5693.061,E2 -5693.061} C_VEL
LIN {X 0,Y 502.422,Z 407.17,A -85,B 0,C 180,E1 -5695.699,E2 -5695.699} C_VEL
LIN {X 0,Y 502.516,Z 403.075,A -85,B 0,C 180,E1 -5698.393,E2 -5698.393} C_VEL
LIN {X 0,Y 502.602,Z 398.508,A -85,B 0,C 180,E1 -5701.463,E2 -5701.463} C_VEL
LIN {X 0,Y 502.697,Z 394.805,A -85,B 0,C 180,E1 -5704.002,E2 -5704.002} C_VEL
LIN {X 0,Y 502.677,Z 393.413,A -85,B 0,C 180,E1 -5704.976,E2 -5704.976} C_VEL
LIN {X 0,Y 502.709,Z 392.864,A -85,B 0,C 180,E1 -5705.957,E2 -5705.957} C_VEL
LIN {X 0,Y 502.804,Z 392.854,A -85,B 0,C 180,E1 -5708.976,E2 -5708.976} C_VEL
LIN {X 0,Y 502.833,Z 392.852,A -85,B 0,C 180,E1 -5712.136,E2 -5712.136} C_VEL
LIN {X 0,Y 502.789,Z 392.857,A -85,B 0,C 180,E1 -5715.47,E2 -5715.47} C_VEL
LIN {X 0,Y 502.823,Z 392.854,A -85,B 0,C 180,E1 -5718.934,E2 -5718.934} C_VEL
LIN {X 0,Y 502.797,Z 392.854,A -85,B 0,C 180,E1 -5722.046,E2 -5722.046} C_VEL
LIN {X 0,Y 502.802,Z 392.853,A -85,B 0,C 180,E1 -5725.034,E2 -5725.034} C_VEL
LIN {X 0,Y 502.786,Z 392.857,A -85,B 0,C 180,E1 -5727.915,E2 -5727.915} C_VEL
LIN {X 0,Y 502.828,Z 392.854,A -85,B 0,C 180,E1 -5730.712,E2 -5730.712} C_VEL
LIN {X 0,Y 502.866,Z 392.843,A -85,B 0,C 180,E1 -5733.439,E2 -5733.439} C_VEL
LIN {X 0,Y 502.78,Z 392.86,A -85,B 0,C 180,E1 -5736.086,E2 -5736.086} C_VEL
LIN {X 0,Y 502.787,Z 392.855,A -85,B 0,C 180,E1 -5738.689,E2 -5738.689} C_VEL
LIN {X 0,Y 502.831,Z 392.851,A -85,B 0,C 180,E1 -5741.248,E2 -5741.248} C_VEL
LIN {X 0,Y 502.852,Z 392.85,A -85,B 0,C 180,E1 -5744.6,E2 -5744.6} C_VEL
LIN {X 0,Y 502.88,Z 392.848,A -85,B 0,C 180,E1 -5748.039,E2 -5748.039} C_VEL
LIN {X 0,Y 502.878,Z 392.844,A -85,B 0,C 180,E1 -5751.157,E2 -5751.157} C_VEL
LIN {X 0,Y 502.932,Z 392.839,A -85,B 0,C 180,E1 -5753.581,E2 -5753.581} C_VEL
LIN {X 0,Y 502.899,Z 392.842,A -85,B 0,C 180,E1 -5756.795,E2 -5756.795} C_VEL
LIN {X 0,Y 503.037,Z 392.823,A -85,B 0,C 180,E1 -5759.199,E2 -5759.199} C_VEL
LIN {X 0,Y 502.905,Z 392.843,A -85,B 0,C 180,E1 -5761.602,E2 -5761.602} C_VEL
LIN {X 0,Y 502.9,Z 392.841,A -85,B 0,C 180,E1 -5763.204,E2 -5763.204} C_VEL
LIN {X 0,Y 502.931,Z 392.838,A -85,B 0,C 180,E1 -5766.419,E2 -5766.419} C_VEL
LIN {X 0,Y 502.878,Z 392.846,A -85,B 0,C 180,E1 -5768.843,E2 -5768.843} C_VEL
LIN {X 0,Y 502.897,Z 392.843,A -85,B 0,C 180,E1 -5772.1,E2 -5772.1} C_VEL
LIN {X 0,Y 502.852,Z 392.851,A -85,B 0,C 180,E1 -5775.4,E2 -5775.4} C_VEL
LIN {X 0,Y 502.85,Z 392.846,A -85,B 0,C 180,E1 -5778.122,E2 -5778.122} C_VEL
LIN {X 0,Y 502.832,Z 392.851,A -85,B 0,C 180,E1 -5780.536,E2 -5780.536} C_VEL
LIN {X 0,Y 502.791,Z 392.854,A -85,B 0,C 180,E1 -5783.041,E2 -5783.041} C_VEL
LIN {X 0,Y 502.825,Z 392.854,A -85,B 0,C 180,E1 -5785.676,E2 -5785.676} C_VEL
LIN {X 0,Y 502.843,Z 392.845,A -85,B 0,C 180,E1 -5788.373,E2 -5788.373} C_VEL
LIN {X 0,Y 502.796,Z 392.854,A -85,B 0,C 180,E1 -5791.499,E2 -5791.499} C_VEL
LIN {X 0,Y 502.807,Z 392.855,A -85,B 0,C 180,E1 -5794.444,E2 -5794.444} C_VEL
LIN {X 0,Y 502.783,Z 392.856,A -85,B 0,C 180,E1 -5797.178,E2 -5797.178} C_VEL
LIN {X 0,Y 502.791,Z 392.854,A -85,B 0,C 180,E1 -5800.015,E2 -5800.015} C_VEL
LIN {X 0,Y 502.805,Z 392.85,A -85,B 0,C 180,E1 -5802.199,E2 -5802.199} C_VEL
LIN {X 0,Y 502.804,Z 392.852,A -85,B 0,C 180,E1 -5805.468,E2 -5805.468} C_VEL
LIN {X 0,Y 502.833,Z 392.855,A -85,B 0,C 180,E1 -5807.864,E2 -5807.864} C_VEL
LIN {X 0,Y 502.804,Z 392.856,A -85,B 0,C 180,E1 -5811.024,E2 -5811.024} C_VEL
LIN {X 0,Y 502.819,Z 392.972,A -85,B 0,C 180,E1 -5812.048,E2 -5812.048} C_VEL
LIN {X 0,Y 503.525,Z 397.333,A -85,B 0,C 180,E1 -5814.111,E2 -5814.111} C_VEL
LIN {X 0,Y 503.486,Z 401.744,A -85,B 0,C 180,E1 -5816.058,E2 -5816.058} C_VEL
LIN {X 0,Y 503.246,Z 408.395,A -85,B 0,C 180,E1 -5818.888,E2 -5818.888} C_VEL
LIN {X 0,Y 503.068,Z 415.129,A -85,B 0,C 180,E1 -5821.658,E2 -5821.658} C_VEL
LIN {X 0,Y 502.853,Z 422.931,A -85,B 0,C 180,E1 -5824.768,E2 -5824.768} C_VEL
LIN {X 0,Y 502.67,Z 430.796,A -85,B 0,C 180,E1 -5827.821,E2 -5827.821} C_VEL
LIN {X 0,Y 502.536,Z 437.536,A -85,B 0,C 180,E1 -5830.388,E2 -5830.388} C_VEL
LIN {X 0,Y 502.406,Z 445.371,A -85,B 0,C 180,E1 -5833.335,E2 -5833.335} C_VEL
LIN {X 0,Y 502.341,Z 451.872,A -85,B 0,C 180,E1 -5835.712,E2 -5835.712} C_VEL
LIN {X 0,Y 504.478,Z 465.032,A -85,B 0,C 180,E1 -5836.095,E2 -5836.095} C_VEL
LIN {X 0,Y 504.382,Z 477.24,A -85,B 0,C 180,E1 -5836.554,E2 -5836.554} C_VEL
LIN {X 0,Y 504.026,Z 489.752,A -85,B 0,C 180,E1 -5837.191,E2 -5837.191} C_VEL
LIN {X 0,Y 503.703,Z 500.78,A -85,B 0,C 180,E1 -5837.919,E2 -5837.919} C_VEL
LIN {X 0,Y 503.354,Z 511.694,A -85,B 0,C 180,E1 -5838.829,E2 -5838.829} C_VEL
LIN {X 0,Y 502.973,Z 520.593,A -85,B 0,C 180,E1 -5839.738,E2 -5839.738} C_VEL
LIN {X 0,Y 502.672,Z 530.265,A -85,B 0,C 180,E1 -5840.95,E2 -5840.95} C_VEL
LIN {X 0,Y 502.432,Z 537.964,A -85,B 0,C 180,E1 -5842.161,E2 -5842.161} C_VEL
LIN {X 0,Y 502.235,Z 545.062,A -85,B 0,C 180,E1 -5843.572,E2 -5843.572} C_VEL
LIN {X 0,Y 502.178,Z 549.785,A -85,B 0,C 180,E1 -5844.781,E2 -5844.781} C_VEL
LIN {X 0,Y 502.144,Z 553.394,A -85,B 0,C 180,E1 -5845.987,E2 -5845.987} C_VEL
LIN {X 0,Y 502.121,Z 555.255,A -85,B 0,C 180,E1 -5846.79,E2 -5846.79} C_VEL
LIN {X 0,Y 502.092,Z 556.65,A -85,B 0,C 180,E1 -5847.593,E2 -5847.593} C_VEL
LIN {X 0,Y 501.99,Z 558.251,A -85,B 0,C 180,E1 -5849.198,E2 -5849.198} C_VEL
LIN {X 0,Y 501.98,Z 558.468,A -85,B 0,C 180,E1 -5850,E2 -5850} C_VEL
LIN {X 0,Y 502.036,Z 557.647,A -85,B 0,C 180,E1 -5851.604,E2 -5851.604} C_VEL
LIN {X 0,Y 502.092,Z 556.653,A -85,B 0,C 180,E1 -5852.407,E2 -5852.407} C_VEL
LIN {X 0,Y 502.12,Z 555.259,A -85,B 0,C 180,E1 -5853.209,E2 -5853.209} C_VEL
LIN {X 0,Y 502.112,Z 552.323,A -85,B 0,C 180,E1 -5854.415,E2 -5854.415} C_VEL
LIN {X 0,Y 502.228,Z 548.353,A -85,B 0,C 180,E1 -5855.621,E2 -5855.621} C_VEL
LIN {X 0,Y 502.332,Z 542.345,A -85,B 0,C 180,E1 -5857.011,E2 -5857.011} C_VEL
LIN {X 0,Y 502.501,Z 535.567,A -85,B 0,C 180,E1 -5858.242,E2 -5858.242} C_VEL
LIN {X 0,Y 502.754,Z 527.284,A -85,B 0,C 180,E1 -5859.454,E2 -5859.454} C_VEL
LIN {X 0,Y 503.042,Z 518.795,A -85,B 0,C 180,E1 -5860.464,E2 -5860.464} C_VEL
LIN {X 0,Y 503.43,Z 508.307,A -85,B 0,C 180,E1 -5861.475,E2 -5861.475} C_VEL
LIN {X 0,Y 503.718,Z 497.005,A -85,B 0,C 180,E1 -5862.351,E2 -5862.351} C_VEL
LIN {X 0,Y 504.126,Z 486.557,A -85,B 0,C 180,E1 -5862.991,E2 -5862.991} C_VEL
LIN {X 0,Y 504.413,Z 474.892,A -85,B 0,C 180,E1 -5863.547,E2 -5863.547} C_VEL
LIN {X 0,Y 504.478,Z 465.028,A -85,B 0,C 180,E1 -5863.905,E2 -5863.905} C_VEL
LIN {X 0,Y 502.311,Z 451.685,A -85,B 0,C 180,E1 -5864.302,E2 -5864.302} C_VEL
LIN {X 0,Y 502.421,Z 444.175,A -85,B 0,C 180,E1 -5867.083,E2 -5867.083} C_VEL
LIN {X 0,Y 502.617,Z 435.26,A -85,B 0,C 180,E1 -5870.471,E2 -5870.471} C_VEL
LIN {X 0,Y 502.747,Z 427.422,A -85,B 0,C 180,E1 -5873.479,E2 -5873.479} C_VEL
LIN {X 0,Y 502.928,Z 419.53,A -85,B 0,C 180,E1 -5876.575,E2 -5876.575} C_VEL
LIN {X 0,Y 503.157,Z 412.846,A -85,B 0,C 180,E1 -5879.267,E2 -5879.267} C_VEL
LIN {X 0,Y 503.377,Z 405.041,A -85,B 0,C 180,E1 -5882.515,E2 -5882.515} C_VEL
LIN {X 0,Y 503.567,Z 398.417,A -85,B 0,C 180,E1 -5885.394,E2 -5885.394} C_VEL
LIN {X 0,Y 503.101,Z 394.464,A -85,B 0,C 180,E1 -5887.226,E2 -5887.226} C_VEL
LIN {X 0,Y 502.807,Z 392.858,A -85,B 0,C 180,E1 -5888.086,E2 -5888.086} C_VEL
LIN {X 0,Y 502.822,Z 392.851,A -85,B 0,C 180,E1 -5891.066,E2 -5891.066} C_VEL
LIN {X 0,Y 502.784,Z 392.858,A -85,B 0,C 180,E1 -5893.376,E2 -5893.376} C_VEL
LIN {X 0,Y 502.792,Z 392.857,A -85,B 0,C 180,E1 -5895.661,E2 -5895.661} C_VEL
LIN {X 0,Y 502.821,Z 392.854,A -85,B 0,C 180,E1 -5899.005,E2 -5899.005} C_VEL
LIN {X 0,Y 502.796,Z 392.855,A -85,B 0,C 180,E1 -5902.046,E2 -5902.046} C_VEL
LIN {X 0,Y 502.81,Z 392.852,A -85,B 0,C 180,E1 -5905.035,E2 -5905.035} C_VEL
LIN {X 0,Y 502.785,Z 392.856,A -85,B 0,C 180,E1 -5907.915,E2 -5907.915} C_VEL
LIN {X 0,Y 502.826,Z 392.853,A -85,B 0,C 180,E1 -5910.712,E2 -5910.712} C_VEL
LIN {X 0,Y 502.865,Z 392.844,A -85,B 0,C 180,E1 -5913.439,E2 -5913.439} C_VEL
LIN {X 0,Y 502.778,Z 392.859,A -85,B 0,C 180,E1 -5916.086,E2 -5916.086} C_VEL
LIN {X 0,Y 502.786,Z 392.855,A -85,B 0,C 180,E1 -5918.689,E2 -5918.689} C_VEL
LIN {X 0,Y 502.833,Z 392.851,A -85,B 0,C 180,E1 -5921.248,E2 -5921.248} C_VEL
LIN {X 0,Y 502.825,Z 392.848,A -85,B 0,C 180,E1 -5923.767,E2 -5923.767} C_VEL
LIN {X 0,Y 502.834,Z 392.852,A -85,B 0,C 180,E1 -5926.255,E2 -5926.255} C_VEL
LIN {X 0,Y 502.894,Z 392.841,A -85,B 0,C 180,E1 -5928.717,E2 -5928.717} C_VEL
LIN {X 0,Y 502.904,Z 392.841,A -85,B 0,C 180,E1 -5931.967,E2 -5931.967} C_VEL
LIN {X 0,Y 502.94,Z 392.837,A -85,B 0,C 180,E1 -5934.387,E2 -5934.387} C_VEL
LIN {X 0,Y 503.026,Z 392.823,A -85,B 0,C 180,E1 -5937.598,E2 -5937.598} C_VEL
LIN {X 0,Y 503.03,Z 392.828,A -85,B 0,C 180,E1 -5940,E2 -5940} C_VEL
LIN {X 0,Y 503.025,Z 392.825,A -85,B 0,C 180,E1 -5942.402,E2 -5942.402} C_VEL
LIN {X 0,Y 502.94,Z 392.837,A -85,B 0,C 180,E1 -5945.614,E2 -5945.614} C_VEL
LIN {X 0,Y 502.905,Z 392.841,A -85,B 0,C 180,E1 -5948.033,E2 -5948.033} C_VEL
LIN {X 0,Y 502.895,Z 392.84,A -85,B 0,C 180,E1 -5951.283,E2 -5951.283} C_VEL
LIN {X 0,Y 502.848,Z 392.846,A -85,B 0,C 180,E1 -5954.571,E2 -5954.571} C_VEL
LIN {X 0,Y 502.825,Z 392.85,A -85,B 0,C 180,E1 -5957.908,E2 -5957.908} C_VEL
LIN {X 0,Y 502.831,Z 392.852,A -85,B 0,C 180,E1 -5960.536,E2 -5960.536} C_VEL
LIN {X 0,Y 502.79,Z 392.854,A -85,B 0,C 180,E1 -5963.041,E2 -5963.041} C_VEL
LIN {X 0,Y 502.824,Z 392.855,A -85,B 0,C 180,E1 -5965.677,E2 -5965.677} C_VEL
LIN {X 0,Y 502.843,Z 392.847,A -85,B 0,C 180,E1 -5968.373,E2 -5968.373} C_VEL
LIN {X 0,Y 502.795,Z 392.854,A -85,B 0,C 180,E1 -5971.499,E2 -5971.499} C_VEL
LIN {X 0,Y 502.809,Z 392.854,A -85,B 0,C 180,E1 -5974.445,E2 -5974.445} C_VEL
LIN {X 0,Y 502.784,Z 392.855,A -85,B 0,C 180,E1 -5977.179,E2 -5977.179} C_VEL
LIN {X 0,Y 502.791,Z 392.853,A -85,B 0,C 180,E1 -5980.015,E2 -5980.015} C_VEL
LIN {X 0,Y 502.805,Z 392.852,A -85,B 0,C 180,E1 -5982.199,E2 -5982.199} C_VEL
LIN {X 0,Y 502.803,Z 392.853,A -85,B 0,C 180,E1 -5985.468,E2 -5985.468} C_VEL
LIN {X 0,Y 502.833,Z 392.852,A -85,B 0,C 180,E1 -5987.864,E2 -5987.864} C_VEL
LIN {X 0,Y 502.803,Z 392.854,A -85,B 0,C 180,E1 -5991.024,E2 -5991.024} C_VEL
LIN {X 0,Y 502.709,Z 392.865,A -85,B 0,C 180,E1 -5994.043,E2 -5994.043} C_VEL
LIN {X 0,Y 502.678,Z 393.279,A -85,B 0,C 180,E1 -5995.025,E2 -5995.025} C_VEL
LIN {X 0,Y 502.675,Z 396.395,A -85,B 0,C 180,E1 -5997.187,E2 -5997.187} C_VEL
LIN {X 0,Y 501.973,Z 397.429,A -85,B 0,C 180,E1 -5997.845,E2 -5997.845} C_VEL
LIN {X 0,Y 499.081,Z 399.318,A -85,B 0,C 180,E1 -5998.909,E2 -5998.909} C_VEL
LIN {X 0,Y 496.639,Z 400.852,A -85,B 0,C 180,E1 -5999.765,E2 -5999.765} C_VEL
LIN {X 0,Y 495.572,Z 401.948,A -85,B 0,C 180,E1 -6000.429,E2 -6000.429} C_VEL
LIN {X 0,Y 495.474,Z 402.29,A -85,B 0,C 180,E1 -6000.654,E2 -6000.654} C_VEL
LIN {X 0,Y 495.409,Z 406.305,A -85,B 0,C 180,E1 -6003.347,E2 -6003.347} C_VEL
LIN {X 0,Y 495.333,Z 409.873,A -85,B 0,C 180,E1 -6005.703,E2 -6005.703} C_VEL
LIN {X 0,Y 495.238,Z 413.958,A -85,B 0,C 180,E1 -6008.348,E2 -6008.348} C_VEL
LIN {X 0,Y 495.188,Z 418.083,A -85,B 0,C 180,E1 -6010.948,E2 -6010.948} C_VEL
LIN {X 0,Y 495.139,Z 422.237,A -85,B 0,C 180,E1 -6013.508,E2 -6013.508} C_VEL
LIN {X 0,Y 495.161,Z 425.681,A -85,B 0,C 180,E1 -6015.566,E2 -6015.566} C_VEL
LIN {X 0,Y 497.744,Z 439.57,A -85,B 0,C 180,E1 -6016.033,E2 -6016.033} C_VEL
LIN {X 0,Y 497.519,Z 451.646,A -85,B 0,C 180,E1 -6016.522,E2 -6016.522} C_VEL
LIN {X 0,Y 497.167,Z 463.399,A -85,B 0,C 180,E1 -6017.159,E2 -6017.159} C_VEL
LIN {X 0,Y 496.827,Z 474.708,A -85,B 0,C 180,E1 -6017.957,E2 -6017.957} C_VEL
LIN {X 0,Y 496.388,Z 485.18,A -85,B 0,C 180,E1 -6018.878,E2 -6018.878} C_VEL
LIN {X 0,Y 496.087,Z 493.734,A -85,B 0,C 180,E1 -6019.8,E2 -6019.8} C_VEL
LIN {X 0,Y 495.77,Z 501.613,A -85,B 0,C 180,E1 -6020.823,E2 -6020.823} C_VEL
LIN {X 0,Y 495.495,Z 509.316,A -85,B 0,C 180,E1 -6022.051,E2 -6022.051} C_VEL
LIN {X 0,Y 495.253,Z 516.38,A -85,B 0,C 180,E1 -6023.481,E2 -6023.481} C_VEL
LIN {X 0,Y 495.128,Z 521.088,A -85,B 0,C 180,E1 -6024.706,E2 -6024.706} C_VEL
LIN {X 0,Y 495.15,Z 524.69,A -85,B 0,C 180,E1 -6025.93,E2 -6025.93} C_VEL
LIN {X 0,Y 495.05,Z 526.556,A -85,B 0,C 180,E1 -6026.745,E2 -6026.745} C_VEL
LIN {X 0,Y 495.025,Z 527.962,A -85,B 0,C 180,E1 -6027.559,E2 -6027.559} C_VEL
LIN {X 0,Y 494.911,Z 529.579,A -85,B 0,C 180,E1 -6029.186,E2 -6029.186} C_VEL
LIN {X 0,Y 494.898,Z 529.816,A -85,B 0,C 180,E1 -6030,E2 -6030} C_VEL
LIN {X 0,Y 494.911,Z 529.631,A -85,B 0,C 180,E1 -6030.814,E2 -6030.814} C_VEL
LIN {X 0,Y 495.025,Z 528.082,A -85,B 0,C 180,E1 -6032.441,E2 -6032.441} C_VEL
LIN {X 0,Y 495.051,Z 526.728,A -85,B 0,C 180,E1 -6033.255,E2 -6033.255} C_VEL
LIN {X 0,Y 495.114,Z 523.866,A -85,B 0,C 180,E1 -6034.478,E2 -6034.478} C_VEL
LIN {X 0,Y 495.234,Z 519.984,A -85,B 0,C 180,E1 -6035.701,E2 -6035.701} C_VEL
LIN {X 0,Y 495.307,Z 514.979,A -85,B 0,C 180,E1 -6036.927,E2 -6036.927} C_VEL
LIN {X 0,Y 495.517,Z 508.674,A -85,B 0,C 180,E1 -6038.154,E2 -6038.154} C_VEL
LIN {X 0,Y 495.758,Z 500.781,A -85,B 0,C 180,E1 -6039.383,E2 -6039.383} C_VEL
LIN {X 0,Y 496.068,Z 492.734,A -85,B 0,C 180,E1 -6040.407,E2 -6040.407} C_VEL
LIN {X 0,Y 496.502,Z 482.911,A -85,B 0,C 180,E1 -6041.43,E2 -6041.43} C_VEL
LIN {X 0,Y 496.868,Z 471.875,A -85,B 0,C 180,E1 -6042.353,E2 -6042.353} C_VEL
LIN {X 0,Y 497.236,Z 461.046,A -85,B 0,C 180,E1 -6043.07,E2 -6043.07} C_VEL
LIN {X 0,Y 497.572,Z 449.092,A -85,B 0,C 180,E1 -6043.685,E2 -6043.685} C_VEL
LIN {X 0,Y 497.618,Z 438.783,A -85,B 0,C 180,E1 -6044.088,E2 -6044.088} C_VEL
LIN {X 0,Y 495.137,Z 425.655,A -85,B 0,C 180,E1 -6044.54,E2 -6044.54} C_VEL
LIN {X 0,Y 495.194,Z 419.88,A -85,B 0,C 180,E1 -6048.029,E2 -6048.029} C_VEL
LIN {X 0,Y 495.203,Z 415.461,A -85,B 0,C 180,E1 -6050.782,E2 -6050.782} C_VEL
LIN {X 0,Y 495.294,Z 411.387,A -85,B 0,C 180,E1 -6053.41,E2 -6053.41} C_VEL
LIN {X 0,Y 495.366,Z 407.298,A -85,B 0,C 180,E1 -6056.092,E2 -6056.092} C_VEL
LIN {X 0,Y 495.455,Z 403.185,A -85,B 0,C 180,E1 -6058.835,E2 -6058.835} C_VEL
LIN {X 0,Y 495.574,Z 398.99,A -85,B 0,C 180,E1 -6061.691,E2 -6061.691} C_VEL
LIN {X 0,Y 495.648,Z 394.718,A -85,B 0,C 180,E1 -6064.673,E2 -6064.673} C_VEL
LIN {X 0,Y 495.618,Z 393.75,A -85,B 0,C 180,E1 -6065.549,E2 -6065.549} C_VEL
LIN {X 0,Y 495.753,Z 393.735,A -85,B 0,C 180,E1 -6068.592,E2 -6068.592} C_VEL
LIN {X 0,Y 495.781,Z 393.729,A -85,B 0,C 180,E1 -6071.779,E2 -6071.779} C_VEL
LIN {X 0,Y 495.74,Z 393.735,A -85,B 0,C 180,E1 -6075.141,E2 -6075.141} C_VEL
LIN {X 0,Y 495.759,Z 393.73,A -85,B 0,C 180,E1 -6078.219,E2 -6078.219} C_VEL
LIN {X 0,Y 495.754,Z 393.729,A -85,B 0,C 180,E1 -6081.408,E2 -6081.408} C_VEL
LIN {X 0,Y 495.751,Z 393.733,A -85,B 0,C 180,E1 -6084.462,E2 -6084.462} C_VEL
LIN {X 0,Y 495.771,Z 393.731,A -85,B 0,C 180,E1 -6087.406,E2 -6087.406} C_VEL
LIN {X 0,Y 495.77,Z 393.729,A -85,B 0,C 180,E1 -6090.254,E2 -6090.254} C_VEL
LIN {X 0,Y 495.827,Z 393.72,A -85,B 0,C 180,E1 -6093.251,E2 -6093.251} C_VEL
LIN {X 0,Y 495.746,Z 393.732,A -85,B 0,C 180,E1 -6096.613,E2 -6096.613} C_VEL
LIN {X 0,Y 495.782,Z 393.729,A -85,B 0,C 180,E1 -6099.324,E2 -6099.324} C_VEL
LIN {X 0,Y 495.785,Z 393.728,A -85,B 0,C 180,E1 -6101.828,E2 -6101.828} C_VEL
LIN {X 0,Y 495.827,Z 393.725,A -85,B 0,C 180,E1 -6104.548,E2 -6104.548} C_VEL
LIN {X 0,Y 495.832,Z 393.725,A -85,B 0,C 180,E1 -6107.965,E2 -6107.965} C_VEL
LIN {X 0,Y 495.847,Z 393.72,A -85,B 0,C 180,E1 -6111.03,E2 -6111.03} C_VEL
LIN {X 0,Y 495.883,Z 393.718,A -85,B 0,C 180,E1 -6113.49,E2 -6113.49} C_VEL
LIN {X 0,Y 495.843,Z 393.721,A -85,B 0,C 180,E1 -6116.75,E2 -6116.75} C_VEL
LIN {X 0,Y 495.874,Z 393.718,A -85,B 0,C 180,E1 -6118.376,E2 -6118.376} C_VEL
LIN {X 0,Y 496.008,Z 393.697,A -85,B 0,C 180,E1 -6120.812,E2 -6120.812} C_VEL
LIN {X 0,Y 495.844,Z 393.721,A -85,B 0,C 180,E1 -6123.25,E2 -6123.25} C_VEL
LIN {X 0,Y 495.883,Z 393.717,A -85,B 0,C 180,E1 -6126.51,E2 -6126.51} C_VEL
LIN {X 0,Y 495.846,Z 393.722,A -85,B 0,C 180,E1 -6128.97,E2 -6128.97} C_VEL
LIN {X 0,Y 495.856,Z 393.719,A -85,B 0,C 180,E1 -6132.275,E2 -6132.275} C_VEL
LIN {X 0,Y 495.811,Z 393.727,A -85,B 0,C 180,E1 -6135.624,E2 -6135.624} C_VEL
LIN {X 0,Y 495.81,Z 393.724,A -85,B 0,C 180,E1 -6138.247,E2 -6138.247} C_VEL
LIN {X 0,Y 495.777,Z 393.731,A -85,B 0,C 180,E1 -6140.756,E2 -6140.756} C_VEL
LIN {X 0,Y 495.746,Z 393.733,A -85,B 0,C 180,E1 -6143.387,E2 -6143.387} C_VEL
LIN {X 0,Y 495.827,Z 393.721,A -85,B 0,C 180,E1 -6146.749,E2 -6146.749} C_VEL
LIN {X 0,Y 495.769,Z 393.728,A -85,B 0,C 180,E1 -6149.746,E2 -6149.746} C_VEL
LIN {X 0,Y 495.77,Z 393.731,A -85,B 0,C 180,E1 -6152.594,E2 -6152.594} C_VEL
LIN {X 0,Y 495.758,Z 393.732,A -85,B 0,C 180,E1 -6155.537,E2 -6155.537} C_VEL
LIN {X 0,Y 495.767,Z 393.729,A -85,B 0,C 180,E1 -6158.768,E2 -6158.768} C_VEL
LIN {X 0,Y 495.76,Z 393.728,A -85,B 0,C 180,E1 -6161.781,E2 -6161.781} C_VEL
LIN {X 0,Y 495.752,Z 393.731,A -85,B 0,C 180,E1 -6165.139,E2 -6165.139} C_VEL
LIN {X 0,Y 495.78,Z 393.733,A -85,B 0,C 180,E1 -6168.221,E2 -6168.221} C_VEL
LIN {X 0,Y 495.754,Z 393.735,A -85,B 0,C 180,E1 -6171.409,E2 -6171.409} C_VEL
LIN {X 0,Y 495.785,Z 393.866,A -85,B 0,C 180,E1 -6171.865,E2 -6171.865} C_VEL
LIN {X 0,Y 496.437,Z 397.889,A -85,B 0,C 180,E1 -6173.798,E2 -6173.798} C_VEL
LIN {X 0,Y 496.478,Z 402.775,A -85,B 0,C 180,E1 -6176.003,E2 -6176.003} C_VEL
LIN {X 0,Y 496.228,Z 409.417,A -85,B 0,C 180,E1 -6178.872,E2 -6178.872} C_VEL
LIN {X 0,Y 496.061,Z 415.577,A -85,B 0,C 180,E1 -6181.449,E2 -6181.449} C_VEL
LIN {X 0,Y 495.797,Z 423.936,A -85,B 0,C 180,E1 -6184.833,E2 -6184.833} C_VEL
LIN {X 0,Y 495.621,Z 431.791,A -85,B 0,C 180,E1 -6187.928,E2 -6187.928} C_VEL
LIN {X 0,Y 495.465,Z 438.494,A -85,B 0,C 180,E1 -6190.528,E2 -6190.528} C_VEL
LIN {X 0,Y 495.339,Z 447.409,A -85,B 0,C 180,E1 -6193.938,E2 -6193.938} C_VEL
LIN {X 0,Y 495.238,Z 451.661,A -85,B 0,C 180,E1 -6195.502,E2 -6195.502} C_VEL
LIN {X 0,Y 497.394,Z 464.822,A -85,B 0,C 180,E1 -6195.893,E2 -6195.893} C_VEL
LIN {X 0,Y 497.657,Z 469.413,A -85,B 0,C 180,E1 -6196.057,E2 -6196.057} C_VEL
LIN {X 0,Y 497.283,Z 482.438,A -85,B 0,C 180,E1 -6196.619,E2 -6196.619} C_VEL
LIN {X 0,Y 496.93,Z 494.053,A -85,B 0,C 180,E1 -6197.291,E2 -6197.291} C_VEL
LIN {X 0,Y 496.576,Z 505.745,A -85,B 0,C 180,E1 -6198.158,E2 -6198.158} C_VEL
LIN {X 0,Y 496.125,Z 516.638,A -85,B 0,C 180,E1 -6199.182,E2 -6199.182} C_VEL
LIN {X 0,Y 495.765,Z 525.49,A -85,B 0,C 180,E1 -6200.206,E2 -6200.206} C_VEL
LIN {X 0,Y 495.497,Z 534.124,A -85,B 0,C 180,E1 -6201.435,E2 -6201.435} C_VEL
LIN {X 0,Y 495.273,Z 541.024,A -85,B 0,C 180,E1 -6202.663,E2 -6202.663} C_VEL
LIN {X 0,Y 495.157,Z 547.068,A -85,B 0,C 180,E1 -6204.018,E2 -6204.018} C_VEL
LIN {X 0,Y 495.016,Z 552.117,A -85,B 0,C 180,E1 -6205.521,E2 -6205.521} C_VEL
LIN {X 0,Y 495.042,Z 555.051,A -85,B 0,C 180,E1 -6206.744,E2 -6206.744} C_VEL
LIN {X 0,Y 494.998,Z 556.446,A -85,B 0,C 180,E1 -6207.559,E2 -6207.559} C_VEL
LIN {X 0,Y 494.963,Z 557.441,A -85,B 0,C 180,E1 -6208.373,E2 -6208.373} C_VEL
LIN {X 0,Y 494.898,Z 558.264,A -85,B 0,C 180,E1 -6210,E2 -6210} C_VEL
LIN {X 0,Y 494.963,Z 557.443,A -85,B 0,C 180,E1 -6211.627,E2 -6211.627} C_VEL
LIN {X 0,Y 494.998,Z 556.449,A -85,B 0,C 180,E1 -6212.441,E2 -6212.441} C_VEL
LIN {X 0,Y 495.042,Z 555.055,A -85,B 0,C 180,E1 -6213.255,E2 -6213.255} C_VEL
LIN {X 0,Y 495.016,Z 552.119,A -85,B 0,C 180,E1 -6214.479,E2 -6214.479} C_VEL
LIN {X 0,Y 495.149,Z 548.148,A -85,B 0,C 180,E1 -6215.702,E2 -6215.702} C_VEL
LIN {X 0,Y 495.257,Z 542.038,A -85,B 0,C 180,E1 -6217.133,E2 -6217.133} C_VEL
LIN {X 0,Y 495.447,Z 535.362,A -85,B 0,C 180,E1 -6218.36,E2 -6218.36} C_VEL
LIN {X 0,Y 495.724,Z 527.079,A -85,B 0,C 180,E1 -6219.589,E2 -6219.589} C_VEL
LIN {X 0,Y 496.027,Z 518.59,A -85,B 0,C 180,E1 -6220.614,E2 -6220.614} C_VEL
LIN {X 0,Y 496.455,Z 508.102,A -85,B 0,C 180,E1 -6221.638,E2 -6221.638} C_VEL
LIN {X 0,Y 496.776,Z 496.673,A -85,B 0,C 180,E1 -6222.536,E2 -6222.536} C_VEL
LIN {X 0,Y 497.185,Z 486.352,A -85,B 0,C 180,E1 -6223.176,E2 -6223.176} C_VEL
LIN {X 0,Y 497.522,Z 474.688,A -85,B 0,C 180,E1 -6223.739,E2 -6223.739} C_VEL
LIN {X 0,Y 497.523,Z 465.587,A -85,B 0,C 180,E1 -6224.077,E2 -6224.077} C_VEL
LIN {X 0,Y 495.335,Z 452.425,A -85,B 0,C 180,E1 -6224.482,E2 -6224.482} C_VEL
LIN {X 0,Y 495.226,Z 451.406,A -85,B 0,C 180,E1 -6224.537,E2 -6224.537} C_VEL
LIN {X 0,Y 495.352,Z 444.027,A -85,B 0,C 180,E1 -6227.334,E2 -6227.334} C_VEL
LIN {X 0,Y 495.571,Z 435.557,A -85,B 0,C 180,E1 -6230.611,E2 -6230.611} C_VEL
LIN {X 0,Y 495.715,Z 427.294,A -85,B 0,C 180,E1 -6233.832,E2 -6233.832} C_VEL
LIN {X 0,Y 495.879,Z 419.955,A -85,B 0,C 180,E1 -6236.761,E2 -6236.761} C_VEL
LIN {X 0,Y 496.133,Z 412.744,A -85,B 0,C 180,E1 -6239.722,E2 -6239.722} C_VEL
LIN {X 0,Y 496.371,Z 406.068,A -85,B 0,C 180,E1 -6242.55,E2 -6242.55} C_VEL
LIN {X 0,Y 496.558,Z 399.449,A -85,B 0,C 180,E1 -6245.471,E2 -6245.471} C_VEL
LIN {X 0,Y 495.982,Z 395.073,A -85,B 0,C 180,E1 -6247.539,E2 -6247.539} C_VEL
LIN {X 0,Y 495.8,Z 393.731,A -85,B 0,C 180,E1 -6248.198,E2 -6248.198} C_VEL
LIN {X 0,Y 495.765,Z 393.73,A -85,B 0,C 180,E1 -6251.294,E2 -6251.294} C_VEL
LIN {X 0,Y 495.739,Z 393.735,A -85,B 0,C 180,E1 -6254,E2 -6254} C_VEL
LIN {X 0,Y 495.727,Z 393.739,A -85,B 0,C 180,E1 -6257.117,E2 -6257.117} C_VEL
LIN {X 0,Y 495.761,Z 393.729,A -85,B 0,C 180,E1 -6259.953,E2 -6259.953} C_VEL
LIN {X 0,Y 495.733,Z 393.737,A -85,B 0,C 180,E1 -6262.553,E2 -6262.553} C_VEL
LIN {X 0,Y 495.786,Z 393.73,A -85,B 0,C 180,E1 -6265.457,E2 -6265.457} C_VEL
LIN {X 0,Y 495.757,Z 393.73,A -85,B 0,C 180,E1 -6268.364,E2 -6268.364} C_VEL
LIN {X 0,Y 495.79,Z 393.724,A -85,B 0,C 180,E1 -6271.507,E2 -6271.507} C_VEL
LIN {X 0,Y 495.782,Z 393.728,A -85,B 0,C 180,E1 -6273.932,E2 -6273.932} C_VEL
LIN {X 0,Y 495.761,Z 393.731,A -85,B 0,C 180,E1 -6277.14,E2 -6277.14} C_VEL
LIN {X 0,Y 495.78,Z 393.728,A -85,B 0,C 180,E1 -6280.11,E2 -6280.11} C_VEL
LIN {X 0,Y 495.789,Z 393.73,A -85,B 0,C 180,E1 -6282.681,E2 -6282.681} C_VEL
LIN {X 0,Y 495.793,Z 393.724,A -85,B 0,C 180,E1 -6285.217,E2 -6285.217} C_VEL
LIN {X 0,Y 495.87,Z 393.717,A -85,B 0,C 180,E1 -6288.555,E2 -6288.555} C_VEL
LIN {X 0,Y 495.876,Z 393.718,A -85,B 0,C 180,E1 -6291.852,E2 -6291.852} C_VEL
LIN {X 0,Y 495.897,Z 393.714,A -85,B 0,C 180,E1 -6294.307,E2 -6294.307} C_VEL
LIN {X 0,Y 495.995,Z 393.699,A -85,B 0,C 180,E1 -6297.564,E2 -6297.564} C_VEL
LIN {X 0,Y 496.001,Z 393.704,A -85,B 0,C 180,E1 -6300,E2 -6300} C_VEL
LIN {X 0,Y 495.994,Z 393.701,A -85,B 0,C 180,E1 -6302.436,E2 -6302.436} C_VEL
LIN {X 0,Y 495.898,Z 393.714,A -85,B 0,C 180,E1 -6305.694,E2 -6305.694} C_VEL
LIN {X 0,Y 495.876,Z 393.717,A -85,B 0,C 180,E1 -6308.148,E2 -6308.148} C_VEL
LIN {X 0,Y 495.876,Z 393.715,A -85,B 0,C 180,E1 -6311.445,E2 -6311.445} C_VEL
LIN {X 0,Y 495.793,Z 393.726,A -85,B 0,C 180,E1 -6314.783,E2 -6314.783} C_VEL
LIN {X 0,Y 495.767,Z 393.732,A -85,B 0,C 180,E1 -6317.319,E2 -6317.319} C_VEL
LIN {X 0,Y 495.78,Z 393.728,A -85,B 0,C 180,E1 -6319.89,E2 -6319.89} C_VEL
LIN {X 0,Y 495.761,Z 393.73,A -85,B 0,C 180,E1 -6322.861,E2 -6322.861} C_VEL
LIN {X 0,Y 495.783,Z 393.728,A -85,B 0,C 180,E1 -6326.068,E2 -6326.068} C_VEL
LIN {X 0,Y 495.774,Z 393.729,A -85,B 0,C 180,E1 -6328.815,E2 -6328.815} C_VEL
LIN {X 0,Y 495.757,Z 393.731,A -85,B 0,C 180,E1 -6331.725,E2 -6331.725} C_VEL
LIN {X 0,Y 495.779,Z 393.729,A -85,B 0,C 180,E1 -6334.695,E2 -6334.695} C_VEL
LIN {X 0,Y 495.735,Z 393.737,A -85,B 0,C 180,E1 -6337.561,E2 -6337.561} C_VEL
LIN {X 0,Y 495.769,Z 393.728,A -85,B 0,C 180,E1 -6340.7,E2 -6340.7} C_VEL
LIN {X 0,Y 495.736,Z 393.734,A -85,B 0,C 180,E1 -6344.001,E2 -6344.001} C_VEL
LIN {X 0,Y 495.736,Z 393.733,A -85,B 0,C 180,E1 -6347.118,E2 -6347.118} C_VEL
LIN {X 0,Y 495.761,Z 393.731,A -85,B 0,C 180,E1 -6349.953,E2 -6349.953} C_VEL
LIN {X 0,Y 495.719,Z 393.734,A -85,B 0,C 180,E1 -6352.555,E2 -6352.555} C_VEL
LIN {X 0,Y 495.645,Z 393.747,A -85,B 0,C 180,E1 -6354.454,E2 -6354.454} C_VEL
LIN {X 0,Y 495.661,Z 394.76,A -85,B 0,C 180,E1 -6355.447,E2 -6355.447} C_VEL
LIN {X 0,Y 495.564,Z 398.921,A -85,B 0,C 180,E1 -6358.35,E2 -6358.35} C_VEL
LIN {X 0,Y 495.474,Z 402.29,A -85,B 0,C 180,E1 -6360.654,E2 -6360.654} C_VEL
LIN {X 0,Y 494.769,Z 403.354,A -85,B 0,C 180,E1 -6361.321,E2 -6361.321} C_VEL
LIN {X 0,Y 491.864,Z 405.269,A -85,B 0,C 180,E1 -6362.4,E2 -6362.4} C_VEL
LIN {X 0,Y 489.423,Z 406.817,A -85,B 0,C 180,E1 -6363.269,E2 -6363.269} C_VEL
LIN {X 0,Y 488.374,Z 407.924,A -85,B 0,C 180,E1 -6363.942,E2 -6363.942} C_VEL
LIN {X 0,Y 488.287,Z 408.272,A -85,B 0,C 180,E1 -6364.17,E2 -6364.17} C_VEL
LIN {X 0,Y 488.222,Z 412.738,A -85,B 0,C 180,E1 -6367.128,E2 -6367.128} C_VEL
LIN {X 0,Y 488.132,Z 416.847,A -85,B 0,C 180,E1 -6369.785,E2 -6369.785} C_VEL
LIN {X 0,Y 488.109,Z 421.006,A -85,B 0,C 180,E1 -6372.4,E2 -6372.4} C_VEL
LIN {X 0,Y 488.046,Z 425.836,A -85,B 0,C 180,E1 -6375.351,E2 -6375.351} C_VEL
LIN {X 0,Y 490.753,Z 439.797,A -85,B 0,C 180,E1 -6375.83,E2 -6375.83} C_VEL
LIN {X 0,Y 490.634,Z 451.864,A -85,B 0,C 180,E1 -6376.329,E2 -6376.329} C_VEL
LIN {X 0,Y 490.235,Z 463.888,A -85,B 0,C 180,E1 -6376.992,E2 -6376.992} C_VEL
LIN {X 0,Y 489.886,Z 474.92,A -85,B 0,C 180,E1 -6377.784,E2 -6377.784} C_VEL
LIN {X 0,Y 489.423,Z 485.391,A -85,B 0,C 180,E1 -6378.717,E2 -6378.717} C_VEL
LIN {X 0,Y 489.108,Z 493.943,A -85,B 0,C 180,E1 -6379.653,E2 -6379.653} C_VEL
LIN {X 0,Y 488.737,Z 501.822,A -85,B 0,C 180,E1 -6380.69,E2 -6380.69} C_VEL
LIN {X 0,Y 488.455,Z 509.523,A -85,B 0,C 180,E1 -6381.936,E2 -6381.936} C_VEL
LIN {X 0,Y 488.183,Z 516.588,A -85,B 0,C 180,E1 -6383.387,E2 -6383.387} C_VEL
LIN {X 0,Y 488.073,Z 521.294,A -85,B 0,C 180,E1 -6384.63,E2 -6384.63} C_VEL
LIN {X 0,Y 488.068,Z 524.896,A -85,B 0,C 180,E1 -6385.871,E2 -6385.871} C_VEL
LIN {X 0,Y 487.979,Z 526.761,A -85,B 0,C 180,E1 -6386.697,E2 -6386.697} C_VEL
LIN {X 0,Y 487.933,Z 528.167,A -85,B 0,C 180,E1 -6387.524,E2 -6387.524} C_VEL
LIN {X 0,Y 487.834,Z 529.783,A -85,B 0,C 180,E1 -6389.175,E2 -6389.175} C_VEL
LIN {X 0,Y 487.819,Z 530.019,A -85,B 0,C 180,E1 -6390,E2 -6390} C_VEL
LIN {X 0,Y 487.834,Z 529.834,A -85,B 0,C 180,E1 -6390.826,E2 -6390.826} C_VEL
LIN {X 0,Y 487.934,Z 528.285,A -85,B 0,C 180,E1 -6392.477,E2 -6392.477} C_VEL
LIN {X 0,Y 487.979,Z 526.93,A -85,B 0,C 180,E1 -6393.303,E2 -6393.303} C_VEL
LIN {X 0,Y 488.012,Z 524.069,A -85,B 0,C 180,E1 -6394.543,E2 -6394.543} C_VEL
LIN {X 0,Y 488.205,Z 519.127,A -85,B 0,C 180,E1 -6396.07,E2 -6396.07} C_VEL
LIN {X 0,Y 488.29,Z 513.209,A -85,B 0,C 180,E1 -6397.443,E2 -6397.443} C_VEL
LIN {X 0,Y 488.593,Z 506.427,A -85,B 0,C 180,E1 -6398.687,E2 -6398.687} C_VEL
LIN {X 0,Y 488.818,Z 499.502,A -85,B 0,C 180,E1 -6399.726,E2 -6399.726} C_VEL
LIN {X 0,Y 489.141,Z 491.159,A -85,B 0,C 180,E1 -6400.765,E2 -6400.765} C_VEL
LIN {X 0,Y 489.672,Z 480.852,A -85,B 0,C 180,E1 -6401.802,E2 -6401.802} C_VEL
LIN {X 0,Y 489.988,Z 470.119,A -85,B 0,C 180,E1 -6402.674,E2 -6402.674} C_VEL
LIN {X 0,Y 490.361,Z 459.479,A -85,B 0,C 180,E1 -6403.362,E2 -6403.362} C_VEL
LIN {X 0,Y 490.744,Z 446.925,A -85,B 0,C 180,E1 -6403.985,E2 -6403.985} C_VEL
LIN {X 0,Y 490.718,Z 439.729,A -85,B 0,C 180,E1 -6404.264,E2 -6404.264} C_VEL
LIN {X 0,Y 488.329,Z 427.466,A -85,B 0,C 180,E1 -6404.688,E2 -6404.688} C_VEL
LIN {X 0,Y 488.062,Z 425.808,A -85,B 0,C 180,E1 -6404.756,E2 -6404.756} C_VEL
LIN {X 0,Y 488.108,Z 420.291,A -85,B 0,C 180,E1 -6408.139,E2 -6408.139} C_VEL
LIN {X 0,Y 488.135,Z 415.604,A -85,B 0,C 180,E1 -6411.097,E2 -6411.097} C_VEL
LIN {X 0,Y 488.246,Z 411.519,A -85,B 0,C 180,E1 -6413.769,E2 -6413.769} C_VEL
LIN {X 0,Y 488.339,Z 406.916,A -85,B 0,C 180,E1 -6416.838,E2 -6416.838} C_VEL
LIN {X 0,Y 488.437,Z 403.296,A -85,B 0,C 180,E1 -6419.289,E2 -6419.289} C_VEL
LIN {X 0,Y 488.556,Z 399.14,A -85,B 0,C 180,E1 -6422.158,E2 -6422.158} C_VEL
LIN {X 0,Y 488.568,Z 394.976,A -85,B 0,C 180,E1 -6425.128,E2 -6425.128} C_VEL
LIN {X 0,Y 488.666,Z 394.615,A -85,B 0,C 180,E1 -6427.16,E2 -6427.16} C_VEL
LIN {X 0,Y 488.721,Z 394.609,A -85,B 0,C 180,E1 -6430.345,E2 -6430.345} C_VEL
LIN {X 0,Y 488.719,Z 394.608,A -85,B 0,C 180,E1 -6432.827,E2 -6432.827} C_VEL
LIN {X 0,Y 488.697,Z 394.612,A -85,B 0,C 180,E1 -6435.977,E2 -6435.977} C_VEL
LIN {X 0,Y 488.71,Z 394.61,A -85,B 0,C 180,E1 -6438.584,E2 -6438.584} C_VEL
LIN {X 0,Y 488.708,Z 394.609,A -85,B 0,C 180,E1 -6440.947,E2 -6440.947} C_VEL
LIN {X 0,Y 488.68,Z 394.613,A -85,B 0,C 180,E1 -6443.868,E2 -6443.868} C_VEL
LIN {X 0,Y 488.742,Z 394.605,A -85,B 0,C 180,E1 -6446.877,E2 -6446.877} C_VEL
LIN {X 0,Y 488.727,Z 394.607,A -85,B 0,C 180,E1 -6449.781,E2 -6449.781} C_VEL
LIN {X 0,Y 488.795,Z 394.597,A -85,B 0,C 180,E1 -6453.056,E2 -6453.056} C_VEL
LIN {X 0,Y 488.684,Z 394.615,A -85,B 0,C 180,E1 -6456.254,E2 -6456.254} C_VEL
LIN {X 0,Y 488.75,Z 394.605,A -85,B 0,C 180,E1 -6459.176,E2 -6459.176} C_VEL
LIN {X 0,Y 488.753,Z 394.605,A -85,B 0,C 180,E1 -6461.631,E2 -6461.631} C_VEL
LIN {X 0,Y 488.766,Z 394.602,A -85,B 0,C 180,E1 -6465,E2 -6465} C_VEL
LIN {X 0,Y 488.809,Z 394.597,A -85,B 0,C 180,E1 -6468.388,E2 -6468.388} C_VEL
LIN {X 0,Y 488.822,Z 394.598,A -85,B 0,C 180,E1 -6471.734,E2 -6471.734} C_VEL
LIN {X 0,Y 488.858,Z 394.591,A -85,B 0,C 180,E1 -6474.224,E2 -6474.224} C_VEL
LIN {X 0,Y 488.963,Z 394.577,A -85,B 0,C 180,E1 -6477.529,E2 -6477.529} C_VEL
LIN {X 0,Y 488.958,Z 394.575,A -85,B 0,C 180,E1 -6480.824,E2 -6480.824} C_VEL
LIN {X 0,Y 488.964,Z 394.575,A -85,B 0,C 180,E1 -6482.471,E2 -6482.471} C_VEL
LIN {X 0,Y 488.858,Z 394.591,A -85,B 0,C 180,E1 -6485.776,E2 -6485.776} C_VEL
LIN {X 0,Y 488.821,Z 394.597,A -85,B 0,C 180,E1 -6488.266,E2 -6488.266} C_VEL
LIN {X 0,Y 488.833,Z 394.595,A -85,B 0,C 180,E1 -6491.612,E2 -6491.612} C_VEL
LIN {X 0,Y 488.766,Z 394.601,A -85,B 0,C 180,E1 -6495,E2 -6495} C_VEL
LIN {X 0,Y 488.758,Z 394.603,A -85,B 0,C 180,E1 -6498.442,E2 -6498.442} C_VEL
LIN {X 0,Y 488.71,Z 394.61,A -85,B 0,C 180,E1 -6501.071,E2 -6501.071} C_VEL
LIN {X 0,Y 488.683,Z 394.615,A -85,B 0,C 180,E1 -6503.746,E2 -6503.746} C_VEL
LIN {X 0,Y 488.795,Z 394.598,A -85,B 0,C 180,E1 -6506.944,E2 -6506.944} C_VEL
LIN {X 0,Y 488.713,Z 394.607,A -85,B 0,C 180,E1 -6510.363,E2 -6510.363} C_VEL
LIN {X 0,Y 488.738,Z 394.605,A -85,B 0,C 180,E1 -6513.484,E2 -6513.484} C_VEL
LIN {X 0,Y 488.69,Z 394.613,A -85,B 0,C 180,E1 -6516.355,E2 -6516.355} C_VEL
LIN {X 0,Y 488.704,Z 394.613,A -85,B 0,C 180,E1 -6519.254,E2 -6519.254} C_VEL
LIN {X 0,Y 488.71,Z 394.607,A -85,B 0,C 180,E1 -6521.6,E2 -6521.6} C_VEL
LIN {X 0,Y 488.715,Z 394.611,A -85,B 0,C 180,E1 -6524.801,E2 -6524.801} C_VEL
LIN {X 0,Y 488.698,Z 394.611,A -85,B 0,C 180,E1 -6527.475,E2 -6527.475} C_VEL
LIN {X 0,Y 488.735,Z 394.611,A -85,B 0,C 180,E1 -6529.677,E2 -6529.677} C_VEL
LIN {X 0,Y 488.775,Z 394.761,A -85,B 0,C 180,E1 -6531.677,E2 -6531.677} C_VEL
LIN {X 0,Y 489.476,Z 399.406,A -85,B 0,C 180,E1 -6533.936,E2 -6533.936} C_VEL
LIN {X 0,Y 489.47,Z 403.8,A -85,B 0,C 180,E1 -6535.946,E2 -6535.946} C_VEL
LIN {X 0,Y 489.219,Z 410.434,A -85,B 0,C 180,E1 -6538.857,E2 -6538.857} C_VEL
LIN {X 0,Y 488.98,Z 417.108,A -85,B 0,C 180,E1 -6541.686,E2 -6541.686} C_VEL
LIN {X 0,Y 488.753,Z 425.049,A -85,B 0,C 180,E1 -6544.946,E2 -6544.946} C_VEL
LIN {X 0,Y 488.542,Z 432.78,A -85,B 0,C 180,E1 -6548.036,E2 -6548.036} C_VEL
LIN {X 0,Y 488.381,Z 439.463,A -85,B 0,C 180,E1 -6550.672,E2 -6550.672} C_VEL
LIN {X 0,Y 488.263,Z 448.304,A -85,B 0,C 180,E1 -6554.128,E2 -6554.128} C_VEL
LIN {X 0,Y 488.175,Z 451.451,A -85,B 0,C 180,E1 -6555.288,E2 -6555.288} C_VEL
LIN {X 0,Y 490.295,Z 464.611,A -85,B 0,C 180,E1 -6555.684,E2 -6555.684} C_VEL
LIN {X 0,Y 490.765,Z 469.209,A -85,B 0,C 180,E1 -6555.857,E2 -6555.857} C_VEL
LIN {X 0,Y 490.365,Z 482.234,A -85,B 0,C 180,E1 -6556.427,E2 -6556.427} C_VEL
LIN {X 0,Y 489.96,Z 494.411,A -85,B 0,C 180,E1 -6557.145,E2 -6557.145} C_VEL
LIN {X 0,Y 489.599,Z 505.54,A -85,B 0,C 180,E1 -6557.986,E2 -6557.986} C_VEL
LIN {X 0,Y 489.138,Z 516.434,A -85,B 0,C 180,E1 -6559.025,E2 -6559.025} C_VEL
LIN {X 0,Y 488.728,Z 525.285,A -85,B 0,C 180,E1 -6560.063,E2 -6560.063} C_VEL
LIN {X 0,Y 488.456,Z 533.919,A -85,B 0,C 180,E1 -6561.311,E2 -6561.311} C_VEL
LIN {X 0,Y 488.204,Z 540.819,A -85,B 0,C 180,E1 -6562.556,E2 -6562.556} C_VEL
LIN {X 0,Y 488.049,Z 546.216,A -85,B 0,C 180,E1 -6563.765,E2 -6563.765} C_VEL
LIN {X 0,Y 487.968,Z 550.688,A -85,B 0,C 180,E1 -6565.042,E2 -6565.042} C_VEL
LIN {X 0,Y 487.934,Z 552.984,A -85,B 0,C 180,E1 -6565.87,E2 -6565.87} C_VEL
LIN {X 0,Y 487.965,Z 554.847,A -85,B 0,C 180,E1 -6566.697,E2 -6566.697} C_VEL
LIN {X 0,Y 487.891,Z 557.238,A -85,B 0,C 180,E1 -6568.349,E2 -6568.349} C_VEL
LIN {X 0,Y 487.819,Z 558.061,A -85,B 0,C 180,E1 -6570,E2 -6570} C_VEL
LIN {X 0,Y 487.891,Z 557.24,A -85,B 0,C 180,E1 -6571.651,E2 -6571.651} C_VEL
LIN {X 0,Y 487.965,Z 554.852,A -85,B 0,C 180,E1 -6573.303,E2 -6573.303} C_VEL
LIN {X 0,Y 487.927,Z 551.915,A -85,B 0,C 180,E1 -6574.544,E2 -6574.544} C_VEL
LIN {X 0,Y 488.052,Z 547.943,A -85,B 0,C 180,E1 -6575.785,E2 -6575.785} C_VEL
LIN {X 0,Y 488.183,Z 541.834,A -85,B 0,C 180,E1 -6577.237,E2 -6577.237} C_VEL
LIN {X 0,Y 488.381,Z 535.157,A -85,B 0,C 180,E1 -6578.482,E2 -6578.482} C_VEL
LIN {X 0,Y 488.691,Z 526.874,A -85,B 0,C 180,E1 -6579.728,E2 -6579.728} C_VEL
LIN {X 0,Y 489.03,Z 518.385,A -85,B 0,C 180,E1 -6580.768,E2 -6580.768} C_VEL
LIN {X 0,Y 489.479,Z 507.897,A -85,B 0,C 180,E1 -6581.806,E2 -6581.806} C_VEL
LIN {X 0,Y 489.845,Z 496.139,A -85,B 0,C 180,E1 -6582.74,E2 -6582.74} C_VEL
LIN {X 0,Y 490.294,Z 484.224,A -85,B 0,C 180,E1 -6583.47,E2 -6583.47} C_VEL
LIN {X 0,Y 490.697,Z 471.879,A -85,B 0,C 180,E1 -6584.039,E2 -6584.039} C_VEL
LIN {X 0,Y 490.6,Z 466.527,A -85,B 0,C 180,E1 -6584.24,E2 -6584.24} C_VEL
LIN {X 0,Y 488.402,Z 453.014,A -85,B 0,C 180,E1 -6584.677,E2 -6584.677} C_VEL
LIN {X 0,Y 488.163,Z 451.265,A -85,B 0,C 180,E1 -6584.726,E2 -6584.726} C_VEL
LIN {X 0,Y 488.298,Z 443.9,A -85,B 0,C 180,E1 -6587.593,E2 -6587.593} C_VEL
LIN {X 0,Y 488.511,Z 435.85,A -85,B 0,C 180,E1 -6590.751,E2 -6590.751} C_VEL
LIN {X 0,Y 488.682,Z 427.164,A -85,B 0,C 180,E1 -6594.197,E2 -6594.197} C_VEL
LIN {X 0,Y 488.846,Z 420.376,A -85,B 0,C 180,E1 -6596.956,E2 -6596.956} C_VEL
LIN {X 0,Y 489.116,Z 413.757,A -85,B 0,C 180,E1 -6599.717,E2 -6599.717} C_VEL
LIN {X 0,Y 489.362,Z 407.092,A -85,B 0,C 180,E1 -6602.586,E2 -6602.586} C_VEL
LIN {X 0,Y 489.544,Z 400.481,A -85,B 0,C 180,E1 -6605.55,E2 -6605.55} C_VEL
LIN {X 0,Y 488.923,Z 395.89,A -85,B 0,C 180,E1 -6607.759,E2 -6607.759} C_VEL
LIN {X 0,Y 488.736,Z 394.611,A -85,B 0,C 180,E1 -6608.457,E2 -6608.457} C_VEL
LIN {X 0,Y 488.725,Z 394.609,A -85,B 0,C 180,E1 -6611.602,E2 -6611.602} C_VEL
LIN {X 0,Y 488.714,Z 394.608,A -85,B 0,C 180,E1 -6614.801,E2 -6614.801} C_VEL
LIN {X 0,Y 488.693,Z 394.611,A -85,B 0,C 180,E1 -6617.474,E2 -6617.474} C_VEL
LIN {X 0,Y 488.734,Z 394.604,A -85,B 0,C 180,E1 -6619.677,E2 -6619.677} C_VEL
LIN {X 0,Y 488.685,Z 394.613,A -85,B 0,C 180,E1 -6622.841,E2 -6622.841} C_VEL
LIN {X 0,Y 488.736,Z 394.607,A -85,B 0,C 180,E1 -6625.887,E2 -6625.887} C_VEL
LIN {X 0,Y 488.694,Z 394.612,A -85,B 0,C 180,E1 -6628.82,E2 -6628.82} C_VEL
LIN {X 0,Y 488.747,Z 394.601,A -85,B 0,C 180,E1 -6631.671,E2 -6631.671} C_VEL
LIN {X 0,Y 488.729,Z 394.61,A -85,B 0,C 180,E1 -6634.443,E2 -6634.443} C_VEL
LIN {X 0,Y 488.723,Z 394.608,A -85,B 0,C 180,E1 -6637.153,E2 -6637.153} C_VEL
LIN {X 0,Y 488.731,Z 394.607,A -85,B 0,C 180,E1 -6639.811,E2 -6639.811} C_VEL
LIN {X 0,Y 488.737,Z 394.606,A -85,B 0,C 180,E1 -6642.423,E2 -6642.423} C_VEL
LIN {X 0,Y 488.764,Z 394.601,A -85,B 0,C 180,E1 -6645,E2 -6645} C_VEL
LIN {X 0,Y 488.832,Z 394.595,A -85,B 0,C 180,E1 -6648.388,E2 -6648.388} C_VEL
LIN {X 0,Y 488.82,Z 394.597,A -85,B 0,C 180,E1 -6651.734,E2 -6651.734} C_VEL
LIN {X 0,Y 488.857,Z 394.591,A -85,B 0,C 180,E1 -6654.224,E2 -6654.224} C_VEL
LIN {X 0,Y 488.962,Z 394.575,A -85,B 0,C 180,E1 -6657.529,E2 -6657.529} C_VEL
LIN {X 0,Y 488.956,Z 394.577,A -85,B 0,C 180,E1 -6660.824,E2 -6660.824} C_VEL
LIN {X 0,Y 488.962,Z 394.577,A -85,B 0,C 180,E1 -6662.471,E2 -6662.471} C_VEL
LIN {X 0,Y 488.857,Z 394.591,A -85,B 0,C 180,E1 -6665.776,E2 -6665.776} C_VEL
LIN {X 0,Y 488.82,Z 394.597,A -85,B 0,C 180,E1 -6668.266,E2 -6668.266} C_VEL
LIN {X 0,Y 488.834,Z 394.593,A -85,B 0,C 180,E1 -6671.612,E2 -6671.612} C_VEL
LIN {X 0,Y 488.764,Z 394.602,A -85,B 0,C 180,E1 -6675,E2 -6675} C_VEL
LIN {X 0,Y 488.749,Z 394.606,A -85,B 0,C 180,E1 -6678.442,E2 -6678.442} C_VEL
LIN {X 0,Y 488.709,Z 394.61,A -85,B 0,C 180,E1 -6681.071,E2 -6681.071} C_VEL
LIN {X 0,Y 488.682,Z 394.614,A -85,B 0,C 180,E1 -6683.746,E2 -6683.746} C_VEL
LIN {X 0,Y 488.794,Z 394.597,A -85,B 0,C 180,E1 -6686.944,E2 -6686.944} C_VEL
LIN {X 0,Y 488.712,Z 394.609,A -85,B 0,C 180,E1 -6690.363,E2 -6690.363} C_VEL
LIN {X 0,Y 488.738,Z 394.605,A -85,B 0,C 180,E1 -6693.485,E2 -6693.485} C_VEL
LIN {X 0,Y 488.692,Z 394.611,A -85,B 0,C 180,E1 -6696.356,E2 -6696.356} C_VEL
LIN {X 0,Y 488.704,Z 394.611,A -85,B 0,C 180,E1 -6699.254,E2 -6699.254} C_VEL
LIN {X 0,Y 488.71,Z 394.609,A -85,B 0,C 180,E1 -6701.6,E2 -6701.6} C_VEL
LIN {X 0,Y 488.714,Z 394.611,A -85,B 0,C 180,E1 -6704.801,E2 -6704.801} C_VEL
LIN {X 0,Y 488.698,Z 394.611,A -85,B 0,C 180,E1 -6707.475,E2 -6707.475} C_VEL
LIN {X 0,Y 488.735,Z 394.608,A -85,B 0,C 180,E1 -6709.677,E2 -6709.677} C_VEL
LIN {X 0,Y 488.665,Z 394.615,A -85,B 0,C 180,E1 -6712.84,E2 -6712.84} C_VEL
LIN {X 0,Y 488.578,Z 394.839,A -85,B 0,C 180,E1 -6714.873,E2 -6714.873} C_VEL
LIN {X 0,Y 488.554,Z 399.014,A -85,B 0,C 180,E1 -6717.842,E2 -6717.842} C_VEL
LIN {X 0,Y 488.436,Z 403.158,A -85,B 0,C 180,E1 -6720.711,E2 -6720.711} C_VEL
LIN {X 0,Y 488.336,Z 407.28,A -85,B 0,C 180,E1 -6723.504,E2 -6723.504} C_VEL
LIN {X 0,Y 488.287,Z 408.272,A -85,B 0,C 180,E1 -6724.17,E2 -6724.17} C_VEL
LIN {X 0,Y 487.613,Z 409.352,A -85,B 0,C 180,E1 -6724.847,E2 -6724.847} C_VEL
LIN {X 0,Y 484.74,Z 411.282,A -85,B 0,C 180,E1 -6725.94,E2 -6725.94} C_VEL
LIN {X 0,Y 482.291,Z 412.845,A -85,B 0,C 180,E1 -6726.821,E2 -6726.821} C_VEL
LIN {X 0,Y 481.21,Z 413.974,A -85,B 0,C 180,E1 -6727.503,E2 -6727.503} C_VEL
LIN {X 0,Y 481.107,Z 414.333,A -85,B 0,C 180,E1 -6727.735,E2 -6727.735} C_VEL
LIN {X 0,Y 481.042,Z 418.391,A -85,B 0,C 180,E1 -6730.365,E2 -6730.365} C_VEL
LIN {X 0,Y 480.985,Z 422.56,A -85,B 0,C 180,E1 -6733.008,E2 -6733.008} C_VEL
LIN {X 0,Y 480.998,Z 426.022,A -85,B 0,C 180,E1 -6735.131,E2 -6735.131} C_VEL
LIN {X 0,Y 483.731,Z 440.024,A -85,B 0,C 180,E1 -6735.62,E2 -6735.62} C_VEL
LIN {X 0,Y 483.935,Z 443.629,A -85,B 0,C 180,E1 -6735.76,E2 -6735.76} C_VEL
LIN {X 0,Y 483.607,Z 456.183,A -85,B 0,C 180,E1 -6736.34,E2 -6736.34} C_VEL
LIN {X 0,Y 483.172,Z 467.768,A -85,B 0,C 180,E1 -6737.048,E2 -6737.048} C_VEL
LIN {X 0,Y 482.837,Z 478.893,A -85,B 0,C 180,E1 -6737.922,E2 -6737.922} C_VEL
LIN {X 0,Y 482.338,Z 488.623,A -85,B 0,C 180,E1 -6738.869,E2 -6738.869} C_VEL
LIN {X 0,Y 481.959,Z 497.471,A -85,B 0,C 180,E1 -6739.922,E2 -6739.922} C_VEL
LIN {X 0,Y 481.59,Z 506.103,A -85,B 0,C 180,E1 -6741.186,E2 -6741.186} C_VEL
LIN {X 0,Y 481.265,Z 512.984,A -85,B 0,C 180,E1 -6742.448,E2 -6742.448} C_VEL
LIN {X 0,Y 481.134,Z 518.205,A -85,B 0,C 180,E1 -6743.636,E2 -6743.636} C_VEL
LIN {X 0,Y 480.91,Z 522.818,A -85,B 0,C 180,E1 -6744.97,E2 -6744.97} C_VEL
LIN {X 0,Y 480.968,Z 525.102,A -85,B 0,C 180,E1 -6745.81,E2 -6745.81} C_VEL
LIN {X 0,Y 480.91,Z 526.966,A -85,B 0,C 180,E1 -6746.649,E2 -6746.649} C_VEL
LIN {X 0,Y 480.846,Z 528.371,A -85,B 0,C 180,E1 -6747.487,E2 -6747.487} C_VEL
LIN {X 0,Y 480.823,Z 529.369,A -85,B 0,C 180,E1 -6748.325,E2 -6748.325} C_VEL
LIN {X 0,Y 480.743,Z 530.223,A -85,B 0,C 180,E1 -6750,E2 -6750} C_VEL
LIN {X 0,Y 480.76,Z 530.037,A -85,B 0,C 180,E1 -6750.838,E2 -6750.838} C_VEL
LIN {X 0,Y 480.824,Z 529.453,A -85,B 0,C 180,E1 -6751.675,E2 -6751.675} C_VEL
LIN {X 0,Y 480.91,Z 527.133,A -85,B 0,C 180,E1 -6753.351,E2 -6753.351} C_VEL
LIN {X 0,Y 480.916,Z 524.272,A -85,B 0,C 180,E1 -6754.61,E2 -6754.61} C_VEL
LIN {X 0,Y 481.129,Z 520.387,A -85,B 0,C 180,E1 -6755.869,E2 -6755.869} C_VEL
LIN {X 0,Y 481.195,Z 515.38,A -85,B 0,C 180,E1 -6757.131,E2 -6757.131} C_VEL
LIN {X 0,Y 481.449,Z 509.075,A -85,B 0,C 180,E1 -6758.394,E2 -6758.394} C_VEL
LIN {X 0,Y 481.76,Z 501.18,A -85,B 0,C 180,E1 -6759.658,E2 -6759.658} C_VEL
LIN {X 0,Y 482.102,Z 493.131,A -85,B 0,C 180,E1 -6760.712,E2 -6760.712} C_VEL
LIN {X 0,Y 482.595,Z 483.305,A -85,B 0,C 180,E1 -6761.764,E2 -6761.764} C_VEL
LIN {X 0,Y 483.022,Z 472.144,A -85,B 0,C 180,E1 -6762.722,E2 -6762.722} C_VEL
LIN {X 0,Y 483.407,Z 461.432,A -85,B 0,C 180,E1 -6763.451,E2 -6763.451} C_VEL
LIN {X 0,Y 483.81,Z 449.472,A -85,B 0,C 180,E1 -6764.082,E2 -6764.082} C_VEL
LIN {X 0,Y 483.831,Z 440.676,A -85,B 0,C 180,E1 -6764.444,E2 -6764.444} C_VEL
LIN {X 0,Y 481.396,Z 427.932,A -85,B 0,C 180,E1 -6764.897,E2 -6764.897} C_VEL
LIN {X 0,Y 481.027,Z 425.992,A -85,B 0,C 180,E1 -6764.977,E2 -6764.977} C_VEL
LIN {X 0,Y 481.052,Z 419.928,A -85,B 0,C 180,E1 -6768.748,E2 -6768.748} C_VEL
LIN {X 0,Y 481.068,Z 415.752,A -85,B 0,C 180,E1 -6771.422,E2 -6771.422} C_VEL
LIN {X 0,Y 481.2,Z 411.663,A -85,B 0,C 180,E1 -6774.139,E2 -6774.139} C_VEL
LIN {X 0,Y 481.279,Z 407.387,A -85,B 0,C 180,E1 -6777.03,E2 -6777.03} C_VEL
LIN {X 0,Y 481.404,Z 403.407,A -85,B 0,C 180,E1 -6779.76,E2 -6779.76} C_VEL
LIN {X 0,Y 481.512,Z 399.251,A -85,B 0,C 180,E1 -6782.687,E2 -6782.687} C_VEL
LIN {X 0,Y 481.517,Z 395.795,A -85,B 0,C 180,E1 -6785.179,E2 -6785.179} C_VEL
LIN {X 0,Y 481.609,Z 395.497,A -85,B 0,C 180,E1 -6786.749,E2 -6786.749} C_VEL
LIN {X 0,Y 481.68,Z 395.484,A -85,B 0,C 180,E1 -6789.94,E2 -6789.94} C_VEL
LIN {X 0,Y 481.668,Z 395.487,A -85,B 0,C 180,E1 -6793.297,E2 -6793.297} C_VEL
LIN {X 0,Y 481.657,Z 395.488,A -85,B 0,C 180,E1 -6795.641,E2 -6795.641} C_VEL
LIN {X 0,Y 481.659,Z 395.489,A -85,B 0,C 180,E1 -6798.958,E2 -6798.958} C_VEL
LIN {X 0,Y 481.658,Z 395.486,A -85,B 0,C 180,E1 -6801.993,E2 -6801.993} C_VEL
LIN {X 0,Y 481.692,Z 395.484,A -85,B 0,C 180,E1 -6805.318,E2 -6805.318} C_VEL
LIN {X 0,Y 481.648,Z 395.489,A -85,B 0,C 180,E1 -6808.312,E2 -6808.312} C_VEL
LIN {X 0,Y 481.703,Z 395.482,A -85,B 0,C 180,E1 -6811.219,E2 -6811.219} C_VEL
LIN {X 0,Y 481.693,Z 395.483,A -85,B 0,C 180,E1 -6814.042,E2 -6814.042} C_VEL
LIN {X 0,Y 481.677,Z 395.484,A -85,B 0,C 180,E1 -6816.812,E2 -6816.812} C_VEL
LIN {X 0,Y 481.701,Z 395.483,A -85,B 0,C 180,E1 -6819.503,E2 -6819.503} C_VEL
LIN {X 0,Y 481.696,Z 395.483,A -85,B 0,C 180,E1 -6822.158,E2 -6822.158} C_VEL
LIN {X 0,Y 481.746,Z 395.477,A -85,B 0,C 180,E1 -6824.776,E2 -6824.776} C_VEL
LIN {X 0,Y 481.754,Z 395.477,A -85,B 0,C 180,E1 -6828.215,E2 -6828.215} C_VEL
LIN {X 0,Y 481.767,Z 395.477,A -85,B 0,C 180,E1 -6831.612,E2 -6831.612} C_VEL
LIN {X 0,Y 481.819,Z 395.467,A -85,B 0,C 180,E1 -6834.14,E2 -6834.14} C_VEL
LIN {X 0,Y 481.93,Z 395.453,A -85,B 0,C 180,E1 -6837.493,E2 -6837.493} C_VEL
LIN {X 0,Y 481.909,Z 395.453,A -85,B 0,C 180,E1 -6840.836,E2 -6840.836} C_VEL
LIN {X 0,Y 481.931,Z 395.451,A -85,B 0,C 180,E1 -6842.507,E2 -6842.507} C_VEL
LIN {X 0,Y 481.819,Z 395.467,A -85,B 0,C 180,E1 -6845.86,E2 -6845.86} C_VEL
LIN {X 0,Y 481.767,Z 395.475,A -85,B 0,C 180,E1 -6848.388,E2 -6848.388} C_VEL
LIN {X 0,Y 481.798,Z 395.473,A -85,B 0,C 180,E1 -6851.784,E2 -6851.784} C_VEL
LIN {X 0,Y 481.746,Z 395.477,A -85,B 0,C 180,E1 -6855.224,E2 -6855.224} C_VEL
LIN {X 0,Y 481.716,Z 395.481,A -85,B 0,C 180,E1 -6858.722,E2 -6858.722} C_VEL
LIN {X 0,Y 481.649,Z 395.489,A -85,B 0,C 180,E1 -6861.395,E2 -6861.395} C_VEL
LIN {X 0,Y 481.664,Z 395.487,A -85,B 0,C 180,E1 -6864.114,E2 -6864.114} C_VEL
LIN {X 0,Y 481.75,Z 395.477,A -85,B 0,C 180,E1 -6867.139,E2 -6867.139} C_VEL
LIN {X 0,Y 481.682,Z 395.483,A -85,B 0,C 180,E1 -6869.741,E2 -6869.741} C_VEL
LIN {X 0,Y 481.675,Z 395.487,A -85,B 0,C 180,E1 -6872.674,E2 -6872.674} C_VEL
LIN {X 0,Y 481.644,Z 395.491,A -85,B 0,C 180,E1 -6875.709,E2 -6875.709} C_VEL
LIN {X 0,Y 481.674,Z 395.485,A -85,B 0,C 180,E1 -6878.859,E2 -6878.859} C_VEL
LIN {X 0,Y 481.655,Z 395.485,A -85,B 0,C 180,E1 -6881.913,E2 -6881.913} C_VEL
LIN {X 0,Y 481.663,Z 395.491,A -85,B 0,C 180,E1 -6884.457,E2 -6884.457} C_VEL
LIN {X 0,Y 481.657,Z 395.493,A -85,B 0,C 180,E1 -6887.84,E2 -6887.84} C_VEL
LIN {X 0,Y 481.699,Z 395.486,A -85,B 0,C 180,E1 -6891.143,E2 -6891.143} C_VEL
LIN {X 0,Y 481.74,Z 395.653,A -85,B 0,C 180,E1 -6891.48,E2 -6891.48} C_VEL
LIN {X 0,Y 482.455,Z 400.432,A -85,B 0,C 180,E1 -6893.845,E2 -6893.845} C_VEL
LIN {X 0,Y 482.532,Z 403.726,A -85,B 0,C 180,E1 -6895.387,E2 -6895.387} C_VEL
LIN {X 0,Y 482.274,Z 410.339,A -85,B 0,C 180,E1 -6898.357,E2 -6898.357} C_VEL
LIN {X 0,Y 482.014,Z 416.999,A -85,B 0,C 180,E1 -6901.239,E2 -6901.239} C_VEL
LIN {X 0,Y 481.703,Z 425.925,A -85,B 0,C 180,E1 -6904.969,E2 -6904.969} C_VEL
LIN {X 0,Y 481.48,Z 433.759,A -85,B 0,C 180,E1 -6908.148,E2 -6908.148} C_VEL
LIN {X 0,Y 481.294,Z 441.526,A -85,B 0,C 180,E1 -6911.261,E2 -6911.261} C_VEL
LIN {X 0,Y 481.119,Z 449.938,A -85,B 0,C 180,E1 -6914.602,E2 -6914.602} C_VEL
LIN {X 0,Y 481.103,Z 451.245,A -85,B 0,C 180,E1 -6915.066,E2 -6915.066} C_VEL
LIN {X 0,Y 483.196,Z 464.401,A -85,B 0,C 180,E1 -6915.469,E2 -6915.469} C_VEL
LIN {X 0,Y 483.872,Z 469.005,A -85,B 0,C 180,E1 -6915.651,E2 -6915.651} C_VEL
LIN {X 0,Y 483.465,Z 482.03,A -85,B 0,C 180,E1 -6916.229,E2 -6916.229} C_VEL
LIN {X 0,Y 483.055,Z 493.231,A -85,B 0,C 180,E1 -6916.892,E2 -6916.892} C_VEL
LIN {X 0,Y 482.645,Z 504.071,A -85,B 0,C 180,E1 -6917.704,E2 -6917.704} C_VEL
LIN {X 0,Y 482.244,Z 514.27,A -85,B 0,C 180,E1 -6918.653,E2 -6918.653} C_VEL
LIN {X 0,Y 481.785,Z 523.446,A -85,B 0,C 180,E1 -6919.706,E2 -6919.706} C_VEL
LIN {X 0,Y 481.429,Z 532.39,A -85,B 0,C 180,E1 -6920.971,E2 -6920.971} C_VEL
LIN {X 0,Y 481.189,Z 539.589,A -85,B 0,C 180,E1 -6922.235,E2 -6922.235} C_VEL
LIN {X 0,Y 480.977,Z 545.425,A -85,B 0,C 180,E1 -6923.522,E2 -6923.522} C_VEL
LIN {X 0,Y 480.9,Z 550.484,A -85,B 0,C 180,E1 -6924.969,E2 -6924.969} C_VEL
LIN {X 0,Y 480.834,Z 552.78,A -85,B 0,C 180,E1 -6925.809,E2 -6925.809} C_VEL
LIN {X 0,Y 480.889,Z 554.644,A -85,B 0,C 180,E1 -6926.649,E2 -6926.649} C_VEL
LIN {X 0,Y 480.792,Z 557.034,A -85,B 0,C 180,E1 -6928.325,E2 -6928.325} C_VEL
LIN {X 0,Y 480.76,Z 557.641,A -85,B 0,C 180,E1 -6929.162,E2 -6929.162} C_VEL
LIN {X 0,Y 480.743,Z 557.857,A -85,B 0,C 180,E1 -6930,E2 -6930} C_VEL
LIN {X 0,Y 480.792,Z 557.036,A -85,B 0,C 180,E1 -6931.675,E2 -6931.675} C_VEL
LIN {X 0,Y 480.889,Z 554.648,A -85,B 0,C 180,E1 -6933.351,E2 -6933.351} C_VEL
LIN {X 0,Y 480.844,Z 551.71,A -85,B 0,C 180,E1 -6934.611,E2 -6934.611} C_VEL
LIN {X 0,Y 480.956,Z 547.738,A -85,B 0,C 180,E1 -6935.871,E2 -6935.871} C_VEL
LIN {X 0,Y 481.112,Z 541.629,A -85,B 0,C 180,E1 -6937.343,E2 -6937.343} C_VEL
LIN {X 0,Y 481.34,Z 534.952,A -85,B 0,C 180,E1 -6938.607,E2 -6938.607} C_VEL
LIN {X 0,Y 481.665,Z 526.669,A -85,B 0,C 180,E1 -6939.872,E2 -6939.872} C_VEL
LIN {X 0,Y 482.045,Z 518.181,A -85,B 0,C 180,E1 -6940.926,E2 -6940.926} C_VEL
LIN {X 0,Y 482.496,Z 507.692,A -85,B 0,C 180,E1 -6941.98,E2 -6941.98} C_VEL
LIN {X 0,Y 482.865,Z 496.605,A -85,B 0,C 180,E1 -6942.877,E2 -6942.877} C_VEL
LIN {X 0,Y 483.323,Z 485.943,A -85,B 0,C 180,E1 -6943.561,E2 -6943.561} C_VEL
LIN {X 0,Y 483.725,Z 474.279,A -85,B 0,C 180,E1 -6944.138,E2 -6944.138} C_VEL
LIN {X 0,Y 483.698,Z 467.467,A -85,B 0,C 180,E1 -6944.408,E2 -6944.408} C_VEL
LIN {X 0,Y 481.522,Z 454.065,A -85,B 0,C 180,E1 -6944.863,E2 -6944.863} C_VEL
LIN {X 0,Y 481.099,Z 451.074,A -85,B 0,C 180,E1 -6944.947,E2 -6944.947} C_VEL
LIN {X 0,Y 481.228,Z 443.739,A -85,B 0,C 180,E1 -6947.86,E2 -6947.86} C_VEL
LIN {X 0,Y 481.461,Z 436.129,A -85,B 0,C 180,E1 -6950.897,E2 -6950.897} C_VEL
LIN {X 0,Y 481.616,Z 428.152,A -85,B 0,C 180,E1 -6954.116,E2 -6954.116} C_VEL
LIN {X 0,Y 481.817,Z 420.796,A -85,B 0,C 180,E1 -6957.155,E2 -6957.155} C_VEL
LIN {X 0,Y 482.163,Z 413.652,A -85,B 0,C 180,E1 -6960.19,E2 -6960.19} C_VEL
LIN {X 0,Y 482.364,Z 407.001,A -85,B 0,C 180,E1 -6963.118,E2 -6963.118} C_VEL
LIN {X 0,Y 482.543,Z 401.511,A -85,B 0,C 180,E1 -6965.632,E2 -6965.632} C_VEL
LIN {X 0,Y 481.872,Z 396.591,A -85,B 0,C 180,E1 -6968.04,E2 -6968.04} C_VEL
LIN {X 0,Y 481.702,Z 395.486,A -85,B 0,C 180,E1 -6968.634,E2 -6968.634} C_VEL
LIN {X 0,Y 481.664,Z 395.491,A -85,B 0,C 180,E1 -6971.914,E2 -6971.914} C_VEL
LIN {X 0,Y 481.662,Z 395.486,A -85,B 0,C 180,E1 -6974.457,E2 -6974.457} C_VEL
LIN {X 0,Y 481.649,Z 395.486,A -85,B 0,C 180,E1 -6977.839,E2 -6977.839} C_VEL
LIN {X 0,Y 481.682,Z 395.487,A -85,B 0,C 180,E1 -6980.651,E2 -6980.651} C_VEL
LIN {X 0,Y 481.633,Z 395.491,A -85,B 0,C 180,E1 -6983.375,E2 -6983.375} C_VEL
LIN {X 0,Y 481.711,Z 395.481,A -85,B 0,C 180,E1 -6986.33,E2 -6986.33} C_VEL
LIN {X 0,Y 481.652,Z 395.488,A -85,B 0,C 180,E1 -6989.417,E2 -6989.417} C_VEL
LIN {X 0,Y 481.702,Z 395.48,A -85,B 0,C 180,E1 -6992.168,E2 -6992.168} C_VEL
LIN {X 0,Y 481.695,Z 395.483,A -85,B 0,C 180,E1 -6994.969,E2 -6994.969} C_VEL
LIN {X 0,Y 481.65,Z 395.489,A -85,B 0,C 180,E1 -6997.705,E2 -6997.705} C_VEL
LIN {X 0,Y 481.71,Z 395.481,A -85,B 0,C 180,E1 -7000.393,E2 -7000.393} C_VEL
LIN {X 0,Y 481.693,Z 395.484,A -85,B 0,C 180,E1 -7003.034,E2 -7003.034} C_VEL
LIN {X 0,Y 481.692,Z 395.481,A -85,B 0,C 180,E1 -7005.639,E2 -7005.639} C_VEL
LIN {X 0,Y 481.797,Z 395.473,A -85,B 0,C 180,E1 -7008.216,E2 -7008.216} C_VEL
LIN {X 0,Y 481.765,Z 395.475,A -85,B 0,C 180,E1 -7011.612,E2 -7011.612} C_VEL
LIN {X 0,Y 481.818,Z 395.467,A -85,B 0,C 180,E1 -7014.14,E2 -7014.14} C_VEL
LIN {X 0,Y 481.929,Z 395.451,A -85,B 0,C 180,E1 -7017.493,E2 -7017.493} C_VEL
LIN {X 0,Y 481.907,Z 395.455,A -85,B 0,C 180,E1 -7020.836,E2 -7020.836} C_VEL
LIN {X 0,Y 481.929,Z 395.453,A -85,B 0,C 180,E1 -7022.507,E2 -7022.507} C_VEL
LIN {X 0,Y 481.819,Z 395.468,A -85,B 0,C 180,E1 -7025.86,E2 -7025.86} C_VEL
LIN {X 0,Y 481.766,Z 395.477,A -85,B 0,C 180,E1 -7028.388,E2 -7028.388} C_VEL
LIN {X 0,Y 481.798,Z 395.471,A -85,B 0,C 180,E1 -7031.784,E2 -7031.784} C_VEL
LIN {X 0,Y 481.745,Z 395.477,A -85,B 0,C 180,E1 -7035.224,E2 -7035.224} C_VEL
LIN {X 0,Y 481.711,Z 395.482,A -85,B 0,C 180,E1 -7038.722,E2 -7038.722} C_VEL
LIN {X 0,Y 481.647,Z 395.488,A -85,B 0,C 180,E1 -7041.395,E2 -7041.395} C_VEL
LIN {X 0,Y 481.663,Z 395.488,A -85,B 0,C 180,E1 -7044.114,E2 -7044.114} C_VEL
LIN {X 0,Y 481.749,Z 395.476,A -85,B 0,C 180,E1 -7047.139,E2 -7047.139} C_VEL
LIN {X 0,Y 481.681,Z 395.485,A -85,B 0,C 180,E1 -7049.741,E2 -7049.741} C_VEL
LIN {X 0,Y 481.674,Z 395.486,A -85,B 0,C 180,E1 -7052.674,E2 -7052.674} C_VEL
LIN {X 0,Y 481.646,Z 395.491,A -85,B 0,C 180,E1 -7055.709,E2 -7055.709} C_VEL
LIN {X 0,Y 481.674,Z 395.483,A -85,B 0,C 180,E1 -7058.859,E2 -7058.859} C_VEL
LIN {X 0,Y 481.655,Z 395.487,A -85,B 0,C 180,E1 -7061.913,E2 -7061.913} C_VEL
LIN {X 0,Y 481.662,Z 395.487,A -85,B 0,C 180,E1 -7064.457,E2 -7064.457} C_VEL
LIN {X 0,Y 481.656,Z 395.49,A -85,B 0,C 180,E1 -7067.84,E2 -7067.84} C_VEL
LIN {X 0,Y 481.682,Z 395.483,A -85,B 0,C 180,E1 -7070.651,E2 -7070.651} C_VEL
LIN {X 0,Y 481.606,Z 395.497,A -85,B 0,C 180,E1 -7073.38,E2 -7073.38} C_VEL
LIN {X 0,Y 481.527,Z 395.662,A -85,B 0,C 180,E1 -7074.819,E2 -7074.819} C_VEL
LIN {X 0,Y 481.51,Z 399.124,A -85,B 0,C 180,E1 -7077.313,E2 -7077.313} C_VEL
LIN {X 0,Y 481.403,Z 403.271,A -85,B 0,C 180,E1 -7080.24,E2 -7080.24} C_VEL
LIN {X 0,Y 481.277,Z 407.403,A -85,B 0,C 180,E1 -7083.084,E2 -7083.084} C_VEL
LIN {X 0,Y 481.195,Z 411.513,A -85,B 0,C 180,E1 -7085.861,E2 -7085.861} C_VEL
LIN {X 0,Y 481.107,Z 414.333,A -85,B 0,C 180,E1 -7087.735,E2 -7087.735} C_VEL
LIN {X 0,Y 480.391,Z 415.442,A -85,B 0,C 180,E1 -7088.421,E2 -7088.421} C_VEL
LIN {X 0,Y 477.494,Z 417.417,A -85,B 0,C 180,E1 -7089.531,E2 -7089.531} C_VEL
LIN {X 0,Y 475.075,Z 419.018,A -85,B 0,C 180,E1 -7090.425,E2 -7090.425} C_VEL
LIN {X 0,Y 474.045,Z 420.184,A -85,B 0,C 180,E1 -7091.118,E2 -7091.118} C_VEL
LIN {X 0,Y 473.965,Z 420.555,A -85,B 0,C 180,E1 -7091.353,E2 -7091.353} C_VEL
LIN {X 0,Y 473.965,Z 426.187,A -85,B 0,C 180,E1 -7094.891,E2 -7094.891} C_VEL
LIN {X 0,Y 476.844,Z 441.015,A -85,B 0,C 180,E1 -7095.436,E2 -7095.436} C_VEL
LIN {X 0,Y 477.045,Z 445.143,A -85,B 0,C 180,E1 -7095.605,E2 -7095.605} C_VEL
LIN {X 0,Y 476.712,Z 456.397,A -85,B 0,C 180,E1 -7096.139,E2 -7096.139} C_VEL
LIN {X 0,Y 476.255,Z 468.524,A -85,B 0,C 180,E1 -7096.894,E2 -7096.894} C_VEL
LIN {X 0,Y 475.891,Z 479.103,A -85,B 0,C 180,E1 -7097.743,E2 -7097.743} C_VEL
LIN {X 0,Y 475.385,Z 488.832,A -85,B 0,C 180,E1 -7098.704,E2 -7098.704} C_VEL
LIN {X 0,Y 474.963,Z 497.68,A -85,B 0,C 180,E1 -7099.772,E2 -7099.772} C_VEL
LIN {X 0,Y 474.565,Z 506.311,A -85,B 0,C 180,E1 -7101.054,E2 -7101.054} C_VEL
LIN {X 0,Y 474.218,Z 513.192,A -85,B 0,C 180,E1 -7102.335,E2 -7102.335} C_VEL
LIN {X 0,Y 474.07,Z 518.741,A -85,B 0,C 180,E1 -7103.628,E2 -7103.628} C_VEL
LIN {X 0,Y 473.851,Z 523.023,A -85,B 0,C 180,E1 -7104.895,E2 -7104.895} C_VEL
LIN {X 0,Y 473.869,Z 525.309,A -85,B 0,C 180,E1 -7105.747,E2 -7105.747} C_VEL
LIN {X 0,Y 473.841,Z 527.171,A -85,B 0,C 180,E1 -7106.599,E2 -7106.599} C_VEL
LIN {X 0,Y 473.763,Z 528.576,A -85,B 0,C 180,E1 -7107.449,E2 -7107.449} C_VEL
LIN {X 0,Y 473.689,Z 530.19,A -85,B 0,C 180,E1 -7109.15,E2 -7109.15} C_VEL
LIN {X 0,Y 473.67,Z 530.426,A -85,B 0,C 180,E1 -7110,E2 -7110} C_VEL
LIN {X 0,Y 473.689,Z 530.24,A -85,B 0,C 180,E1 -7110.85,E2 -7110.85} C_VEL
LIN {X 0,Y 473.763,Z 528.691,A -85,B 0,C 180,E1 -7112.551,E2 -7112.551} C_VEL
LIN {X 0,Y 473.842,Z 527.335,A -85,B 0,C 180,E1 -7113.401,E2 -7113.401} C_VEL
LIN {X 0,Y 473.826,Z 524.475,A -85,B 0,C 180,E1 -7114.679,E2 -7114.679} C_VEL
LIN {X 0,Y 474.072,Z 520.588,A -85,B 0,C 180,E1 -7115.957,E2 -7115.957} C_VEL
LIN {X 0,Y 474.145,Z 515.581,A -85,B 0,C 180,E1 -7117.238,E2 -7117.238} C_VEL
LIN {X 0,Y 474.42,Z 509.276,A -85,B 0,C 180,E1 -7118.519,E2 -7118.519} C_VEL
LIN {X 0,Y 474.739,Z 501.38,A -85,B 0,C 180,E1 -7119.802,E2 -7119.802} C_VEL
LIN {X 0,Y 475.13,Z 493.33,A -85,B 0,C 180,E1 -7120.871,E2 -7120.871} C_VEL
LIN {X 0,Y 475.651,Z 483.504,A -85,B 0,C 180,E1 -7121.938,E2 -7121.938} C_VEL
LIN {X 0,Y 476.05,Z 473.838,A -85,B 0,C 180,E1 -7122.794,E2 -7122.794} C_VEL
LIN {X 0,Y 476.451,Z 463.348,A -85,B 0,C 180,E1 -7123.545,E2 -7123.545} C_VEL
LIN {X 0,Y 476.902,Z 450.792,A -85,B 0,C 180,E1 -7124.236,E2 -7124.236} C_VEL
LIN {X 0,Y 476.929,Z 441.642,A -85,B 0,C 180,E1 -7124.63,E2 -7124.63} C_VEL
LIN {X 0,Y 474.617,Z 429.501,A -85,B 0,C 180,E1 -7125.082,E2 -7125.082} C_VEL
LIN {X 0,Y 473.977,Z 426.182,A -85,B 0,C 180,E1 -7125.202,E2 -7125.202} C_VEL
LIN {X 0,Y 473.973,Z 420.089,A -85,B 0,C 180,E1 -7129.039,E2 -7129.039} C_VEL
LIN {X 0,Y 474.014,Z 415.904,A -85,B 0,C 180,E1 -7131.757,E2 -7131.757} C_VEL
LIN {X 0,Y 474.133,Z 411.798,A -85,B 0,C 180,E1 -7134.522,E2 -7134.522} C_VEL
LIN {X 0,Y 474.24,Z 407.682,A -85,B 0,C 180,E1 -7137.349,E2 -7137.349} C_VEL
LIN {X 0,Y 474.366,Z 403.521,A -85,B 0,C 180,E1 -7140.247,E2 -7140.247} C_VEL
LIN {X 0,Y 474.475,Z 399.341,A -85,B 0,C 180,E1 -7143.234,E2 -7143.234} C_VEL
LIN {X 0,Y 474.469,Z 396.386,A -85,B 0,C 180,E1 -7145.444,E2 -7145.444} C_VEL
LIN {X 0,Y 474.613,Z 396.368,A -85,B 0,C 180,E1 -7148.457,E2 -7148.457} C_VEL
LIN {X 0,Y 474.635,Z 396.362,A -85,B 0,C 180,E1 -7150.96,E2 -7150.96} C_VEL
LIN {X 0,Y 474.615,Z 396.366,A -85,B 0,C 180,E1 -7154.105,E2 -7154.105} C_VEL
LIN {X 0,Y 474.609,Z 396.368,A -85,B 0,C 180,E1 -7157.065,E2 -7157.065} C_VEL
LIN {X 0,Y 474.631,Z 396.363,A -85,B 0,C 180,E1 -7160.352,E2 -7160.352} C_VEL
LIN {X 0,Y 474.592,Z 396.367,A -85,B 0,C 180,E1 -7163.677,E2 -7163.677} C_VEL
LIN {X 0,Y 474.646,Z 396.361,A -85,B 0,C 180,E1 -7166.78,E2 -7166.78} C_VEL
LIN {X 0,Y 474.608,Z 396.366,A -85,B 0,C 180,E1 -7169.77,E2 -7169.77} C_VEL
LIN {X 0,Y 474.7,Z 396.356,A -85,B 0,C 180,E1 -7172.68,E2 -7172.68} C_VEL
LIN {X 0,Y 474.644,Z 396.359,A -85,B 0,C 180,E1 -7175.506,E2 -7175.506} C_VEL
LIN {X 0,Y 474.674,Z 396.358,A -85,B 0,C 180,E1 -7179.185,E2 -7179.185} C_VEL
LIN {X 0,Y 474.65,Z 396.361,A -85,B 0,C 180,E1 -7181.884,E2 -7181.884} C_VEL
LIN {X 0,Y 474.703,Z 396.356,A -85,B 0,C 180,E1 -7184.544,E2 -7184.544} C_VEL
LIN {X 0,Y 474.708,Z 396.357,A -85,B 0,C 180,E1 -7188.038,E2 -7188.038} C_VEL
LIN {X 0,Y 474.732,Z 396.352,A -85,B 0,C 180,E1 -7191.486,E2 -7191.486} C_VEL
LIN {X 0,Y 474.782,Z 396.344,A -85,B 0,C 180,E1 -7194.052,E2 -7194.052} C_VEL
LIN {X 0,Y 474.896,Z 396.329,A -85,B 0,C 180,E1 -7197.455,E2 -7197.455} C_VEL
LIN {X 0,Y 474.915,Z 396.331,A -85,B 0,C 180,E1 -7200,E2 -7200} C_VEL
LIN {X 0,Y 474.897,Z 396.327,A -85,B 0,C 180,E1 -7202.545,E2 -7202.545} C_VEL
LIN {X 0,Y 474.782,Z 396.344,A -85,B 0,C 180,E1 -7205.948,E2 -7205.948} C_VEL
LIN {X 0,Y 474.732,Z 396.351,A -85,B 0,C 180,E1 -7208.513,E2 -7208.513} C_VEL
LIN {X 0,Y 474.743,Z 396.351,A -85,B 0,C 180,E1 -7211.961,E2 -7211.961} C_VEL
LIN {X 0,Y 474.684,Z 396.357,A -85,B 0,C 180,E1 -7215.768,E2 -7215.768} C_VEL
LIN {X 0,Y 474.669,Z 396.36,A -85,B 0,C 180,E1 -7219.01,E2 -7219.01} C_VEL
LIN {X 0,Y 474.591,Z 396.369,A -85,B 0,C 180,E1 -7221.729,E2 -7221.729} C_VEL
LIN {X 0,Y 474.644,Z 396.361,A -85,B 0,C 180,E1 -7224.494,E2 -7224.494} C_VEL
LIN {X 0,Y 474.702,Z 396.357,A -85,B 0,C 180,E1 -7227.339,E2 -7227.339} C_VEL
LIN {X 0,Y 474.607,Z 396.367,A -85,B 0,C 180,E1 -7230.81,E2 -7230.81} C_VEL
LIN {X 0,Y 474.641,Z 396.362,A -85,B 0,C 180,E1 -7233.984,E2 -7233.984} C_VEL
LIN {X 0,Y 474.577,Z 396.37,A -85,B 0,C 180,E1 -7236.9,E2 -7236.9} C_VEL
LIN {X 0,Y 474.63,Z 396.363,A -85,B 0,C 180,E1 -7239.648,E2 -7239.648} C_VEL
LIN {X 0,Y 474.618,Z 396.368,A -85,B 0,C 180,E1 -7242.934,E2 -7242.934} C_VEL
LIN {X 0,Y 474.618,Z 396.365,A -85,B 0,C 180,E1 -7245.896,E2 -7245.896} C_VEL
LIN {X 0,Y 474.635,Z 396.364,A -85,B 0,C 180,E1 -7249.04,E2 -7249.04} C_VEL
LIN {X 0,Y 474.681,Z 396.545,A -85,B 0,C 180,E1 -7251.278,E2 -7251.278} C_VEL
LIN {X 0,Y 475.45,Z 401.453,A -85,B 0,C 180,E1 -7253.753,E2 -7253.753} C_VEL
LIN {X 0,Y 475.478,Z 405.923,A -85,B 0,C 180,E1 -7255.867,E2 -7255.867} C_VEL
LIN {X 0,Y 475.163,Z 413.019,A -85,B 0,C 180,E1 -7259.078,E2 -7259.078} C_VEL
LIN {X 0,Y 474.906,Z 419.108,A -85,B 0,C 180,E1 -7261.734,E2 -7261.734} C_VEL
LIN {X 0,Y 474.654,Z 426.909,A -85,B 0,C 180,E1 -7265.04,E2 -7265.04} C_VEL
LIN {X 0,Y 474.422,Z 434.732,A -85,B 0,C 180,E1 -7268.263,E2 -7268.263} C_VEL
LIN {X 0,Y 474.214,Z 442.749,A -85,B 0,C 180,E1 -7271.532,E2 -7271.532} C_VEL
LIN {X 0,Y 474.028,Z 450.884,A -85,B 0,C 180,E1 -7274.825,E2 -7274.825} C_VEL
LIN {X 0,Y 476.319,Z 465.348,A -85,B 0,C 180,E1 -7275.296,E2 -7275.296} C_VEL
LIN {X 0,Y 476.946,Z 470.177,A -85,B 0,C 180,E1 -7275.493,E2 -7275.493} C_VEL
LIN {X 0,Y 476.576,Z 481.828,A -85,B 0,C 180,E1 -7276.026,E2 -7276.026} C_VEL
LIN {X 0,Y 476.092,Z 494.144,A -85,B 0,C 180,E1 -7276.773,E2 -7276.773} C_VEL
LIN {X 0,Y 475.697,Z 503.444,A -85,B 0,C 180,E1 -7277.486,E2 -7277.486} C_VEL
LIN {X 0,Y 475.263,Z 514.066,A -85,B 0,C 180,E1 -7278.484,E2 -7278.484} C_VEL
LIN {X 0,Y 474.776,Z 523.242,A -85,B 0,C 180,E1 -7279.552,E2 -7279.552} C_VEL
LIN {X 0,Y 474.385,Z 532.185,A -85,B 0,C 180,E1 -7280.836,E2 -7280.836} C_VEL
LIN {X 0,Y 474.108,Z 539.384,A -85,B 0,C 180,E1 -7282.119,E2 -7282.119} C_VEL
LIN {X 0,Y 473.879,Z 545.69,A -85,B 0,C 180,E1 -7283.548,E2 -7283.548} C_VEL
LIN {X 0,Y 473.832,Z 550.28,A -85,B 0,C 180,E1 -7284.894,E2 -7284.894} C_VEL
LIN {X 0,Y 473.74,Z 552.575,A -85,B 0,C 180,E1 -7285.746,E2 -7285.746} C_VEL
LIN {X 0,Y 473.797,Z 554.44,A -85,B 0,C 180,E1 -7286.598,E2 -7286.598} C_VEL
LIN {X 0,Y 473.741,Z 555.835,A -85,B 0,C 180,E1 -7287.449,E2 -7287.449} C_VEL
LIN {X 0,Y 473.688,Z 557.438,A -85,B 0,C 180,E1 -7289.15,E2 -7289.15} C_VEL
LIN {X 0,Y 473.669,Z 557.654,A -85,B 0,C 180,E1 -7290,E2 -7290} C_VEL
LIN {X 0,Y 473.688,Z 557.439,A -85,B 0,C 180,E1 -7290.85,E2 -7290.85} C_VEL
LIN {X 0,Y 473.741,Z 555.838,A -85,B 0,C 180,E1 -7292.551,E2 -7292.551} C_VEL
LIN {X 0,Y 473.797,Z 554.444,A -85,B 0,C 180,E1 -7293.401,E2 -7293.401} C_VEL
LIN {X 0,Y 473.767,Z 551.506,A -85,B 0,C 180,E1 -7294.68,E2 -7294.68} C_VEL
LIN {X 0,Y 473.864,Z 547.533,A -85,B 0,C 180,E1 -7295.959,E2 -7295.959} C_VEL
LIN {X 0,Y 474.032,Z 541.424,A -85,B 0,C 180,E1 -7297.454,E2 -7297.454} C_VEL
LIN {X 0,Y 474.301,Z 534.747,A -85,B 0,C 180,E1 -7298.736,E2 -7298.736} C_VEL
LIN {X 0,Y 474.616,Z 526.463,A -85,B 0,C 180,E1 -7300.02,E2 -7300.02} C_VEL
LIN {X 0,Y 475.051,Z 517.976,A -85,B 0,C 180,E1 -7301.088,E2 -7301.088} C_VEL
LIN {X 0,Y 475.505,Z 507.688,A -85,B 0,C 180,E1 -7302.14,E2 -7302.14} C_VEL
LIN {X 0,Y 475.956,Z 496.11,A -85,B 0,C 180,E1 -7303.089,E2 -7303.089} C_VEL
LIN {X 0,Y 476.482,Z 483.814,A -85,B 0,C 180,E1 -7303.868,E2 -7303.868} C_VEL
LIN {X 0,Y 476.929,Z 471.468,A -85,B 0,C 180,E1 -7304.453,E2 -7304.453} C_VEL
LIN {X 0,Y 476.358,Z 465.718,A -85,B 0,C 180,E1 -7304.689,E2 -7304.689} C_VEL
LIN {X 0,Y 474.233,Z 452.353,A -85,B 0,C 180,E1 -7305.13,E2 -7305.13} C_VEL
LIN {X 0,Y 474.037,Z 450.883,A -85,B 0,C 180,E1 -7305.175,E2 -7305.175} C_VEL
LIN {X 0,Y 474.213,Z 442.747,A -85,B 0,C 180,E1 -7308.467,E2 -7308.467} C_VEL
LIN {X 0,Y 474.386,Z 436.427,A -85,B 0,C 180,E1 -7311.038,E2 -7311.038} C_VEL
LIN {X 0,Y 474.605,Z 428.01,A -85,B 0,C 180,E1 -7314.496,E2 -7314.496} C_VEL
LIN {X 0,Y 474.859,Z 420.201,A -85,B 0,C 180,E1 -7317.788,E2 -7317.788} C_VEL
LIN {X 0,Y 475.14,Z 414.653,A -85,B 0,C 180,E1 -7320.193,E2 -7320.193} C_VEL
LIN {X 0,Y 475.362,Z 408.019,A -85,B 0,C 180,E1 -7323.163,E2 -7323.163} C_VEL
LIN {X 0,Y 475.538,Z 402.716,A -85,B 0,C 180,E1 -7325.625,E2 -7325.625} C_VEL
LIN {X 0,Y 474.824,Z 397.29,A -85,B 0,C 180,E1 -7328.328,E2 -7328.328} C_VEL
LIN {X 0,Y 474.667,Z 396.362,A -85,B 0,C 180,E1 -7328.859,E2 -7328.859} C_VEL
LIN {X 0,Y 474.633,Z 396.367,A -85,B 0,C 180,E1 -7332.238,E2 -7332.238} C_VEL
LIN {X 0,Y 474.623,Z 396.368,A -85,B 0,C 180,E1 -7335.297,E2 -7335.297} C_VEL
LIN {X 0,Y 474.622,Z 396.361,A -85,B 0,C 180,E1 -7338.215,E2 -7338.215} C_VEL
LIN {X 0,Y 474.646,Z 396.361,A -85,B 0,C 180,E1 -7340.454,E2 -7340.454} C_VEL
LIN {X 0,Y 474.595,Z 396.368,A -85,B 0,C 180,E1 -7343.677,E2 -7343.677} C_VEL
LIN {X 0,Y 474.644,Z 396.361,A -85,B 0,C 180,E1 -7346.78,E2 -7346.78} C_VEL
LIN {X 0,Y 474.607,Z 396.364,A -85,B 0,C 180,E1 -7349.77,E2 -7349.77} C_VEL
LIN {X 0,Y 474.699,Z 396.358,A -85,B 0,C 180,E1 -7352.68,E2 -7352.68} C_VEL
LIN {X 0,Y 474.643,Z 396.362,A -85,B 0,C 180,E1 -7355.506,E2 -7355.506} C_VEL
LIN {X 0,Y 474.673,Z 396.36,A -85,B 0,C 180,E1 -7359.185,E2 -7359.185} C_VEL
LIN {X 0,Y 474.659,Z 396.358,A -85,B 0,C 180,E1 -7361.884,E2 -7361.884} C_VEL
LIN {X 0,Y 474.702,Z 396.358,A -85,B 0,C 180,E1 -7364.544,E2 -7364.544} C_VEL
LIN {X 0,Y 474.741,Z 396.351,A -85,B 0,C 180,E1 -7368.039,E2 -7368.039} C_VEL
LIN {X 0,Y 474.73,Z 396.351,A -85,B 0,C 180,E1 -7371.487,E2 -7371.487} C_VEL
LIN {X 0,Y 474.781,Z 396.344,A -85,B 0,C 180,E1 -7374.052,E2 -7374.052} C_VEL
LIN {X 0,Y 474.895,Z 396.328,A -85,B 0,C 180,E1 -7377.455,E2 -7377.455} C_VEL
LIN {X 0,Y 474.914,Z 396.33,A -85,B 0,C 180,E1 -7380,E2 -7380} C_VEL
LIN {X 0,Y 474.895,Z 396.33,A -85,B 0,C 180,E1 -7382.545,E2 -7382.545} C_VEL
LIN {X 0,Y 474.781,Z 396.344,A -85,B 0,C 180,E1 -7385.948,E2 -7385.948} C_VEL
LIN {X 0,Y 474.731,Z 396.352,A -85,B 0,C 180,E1 -7388.514,E2 -7388.514} C_VEL
LIN {X 0,Y 474.741,Z 396.353,A -85,B 0,C 180,E1 -7391.962,E2 -7391.962} C_VEL
LIN {X 0,Y 474.682,Z 396.358,A -85,B 0,C 180,E1 -7395.768,E2 -7395.768} C_VEL
LIN {X 0,Y 474.666,Z 396.359,A -85,B 0,C 180,E1 -7399.01,E2 -7399.01} C_VEL
LIN {X 0,Y 474.59,Z 396.368,A -85,B 0,C 180,E1 -7401.729,E2 -7401.729} C_VEL
LIN {X 0,Y 474.643,Z 396.359,A -85,B 0,C 180,E1 -7404.494,E2 -7404.494} C_VEL
LIN {X 0,Y 474.701,Z 396.355,A -85,B 0,C 180,E1 -7407.339,E2 -7407.339} C_VEL
LIN {X 0,Y 474.606,Z 396.366,A -85,B 0,C 180,E1 -7410.81,E2 -7410.81} C_VEL
LIN {X 0,Y 474.641,Z 396.364,A -85,B 0,C 180,E1 -7413.984,E2 -7413.984} C_VEL
LIN {X 0,Y 474.578,Z 396.368,A -85,B 0,C 180,E1 -7416.9,E2 -7416.9} C_VEL
LIN {X 0,Y 474.63,Z 396.364,A -85,B 0,C 180,E1 -7419.648,E2 -7419.648} C_VEL
LIN {X 0,Y 474.617,Z 396.366,A -85,B 0,C 180,E1 -7422.934,E2 -7422.934} C_VEL
LIN {X 0,Y 474.617,Z 396.367,A -85,B 0,C 180,E1 -7425.896,E2 -7425.896} C_VEL
LIN {X 0,Y 474.634,Z 396.362,A -85,B 0,C 180,E1 -7429.04,E2 -7429.04} C_VEL
LIN {X 0,Y 474.609,Z 396.368,A -85,B 0,C 180,E1 -7431.705,E2 -7431.705} C_VEL
LIN {X 0,Y 474.471,Z 396.415,A -85,B 0,C 180,E1 -7434.713,E2 -7434.713} C_VEL
LIN {X 0,Y 474.453,Z 400.367,A -85,B 0,C 180,E1 -7437.601,E2 -7437.601} C_VEL
LIN {X 0,Y 474.34,Z 404.768,A -85,B 0,C 180,E1 -7440.729,E2 -7440.729} C_VEL
LIN {X 0,Y 474.207,Z 408.912,A -85,B 0,C 180,E1 -7443.601,E2 -7443.601} C_VEL
LIN {X 0,Y 474.124,Z 413.581,A -85,B 0,C 180,E1 -7446.786,E2 -7446.786} C_VEL
LIN {X 0,Y 473.963,Z 418.549,A -85,B 0,C 180,E1 -7450.059,E2 -7450.059} C_VEL
LIN {X 0,Y 473.965,Z 420.555,A -85,B 0,C 180,E1 -7451.353,E2 -7451.353} C_VEL
LIN {X 0,Y 473.28,Z 421.337,A -85,B 0,C 180,E1 -7451.816,E2 -7451.816} C_VEL
LIN {X 0,Y 470.392,Z 422.715,A -85,B 0,C 180,E1 -7452.535,E2 -7452.535} C_VEL
LIN {X 0,Y 467.495,Z 424.107,A -85,B 0,C 180,E1 -7453.263,E2 -7453.263} C_VEL
LIN {X 0,Y 466.817,Z 424.912,A -85,B 0,C 180,E1 -7453.735,E2 -7453.735} C_VEL
LIN {X 0,Y 466.904,Z 426.394,A -85,B 0,C 180,E1 -7454.666,E2 -7454.666} C_VEL
LIN {X 0,Y 469.809,Z 440.862,A -85,B 0,C 180,E1 -7455.199,E2 -7455.199} C_VEL
LIN {X 0,Y 470.183,Z 445.359,A -85,B 0,C 180,E1 -7455.39,E2 -7455.39} C_VEL
LIN {X 0,Y 469.832,Z 456.609,A -85,B 0,C 180,E1 -7455.932,E2 -7455.932} C_VEL
LIN {X 0,Y 469.354,Z 468.409,A -85,B 0,C 180,E1 -7456.675,E2 -7456.675} C_VEL
LIN {X 0,Y 468.944,Z 479.313,A -85,B 0,C 180,E1 -7457.559,E2 -7457.559} C_VEL
LIN {X 0,Y 468.429,Z 489.041,A -85,B 0,C 180,E1 -7458.534,E2 -7458.534} C_VEL
LIN {X 0,Y 467.982,Z 497.888,A -85,B 0,C 180,E1 -7459.618,E2 -7459.618} C_VEL
LIN {X 0,Y 467.543,Z 506.519,A -85,B 0,C 180,E1 -7460.919,E2 -7460.919} C_VEL
LIN {X 0,Y 467.188,Z 513.398,A -85,B 0,C 180,E1 -7462.219,E2 -7462.219} C_VEL
LIN {X 0,Y 467.006,Z 519.273,A -85,B 0,C 180,E1 -7463.62,E2 -7463.62} C_VEL
LIN {X 0,Y 466.796,Z 523.229,A -85,B 0,C 180,E1 -7464.817,E2 -7464.817} C_VEL
LIN {X 0,Y 466.771,Z 525.515,A -85,B 0,C 180,E1 -7465.683,E2 -7465.683} C_VEL
LIN {X 0,Y 466.774,Z 527.375,A -85,B 0,C 180,E1 -7466.547,E2 -7466.547} C_VEL
LIN {X 0,Y 466.684,Z 528.78,A -85,B 0,C 180,E1 -7467.411,E2 -7467.411} C_VEL
LIN {X 0,Y 466.62,Z 530.394,A -85,B 0,C 180,E1 -7469.137,E2 -7469.137} C_VEL
LIN {X 0,Y 466.599,Z 530.629,A -85,B 0,C 180,E1 -7470,E2 -7470} C_VEL
LIN {X 0,Y 466.62,Z 530.443,A -85,B 0,C 180,E1 -7470.863,E2 -7470.863} C_VEL
LIN {X 0,Y 466.684,Z 528.893,A -85,B 0,C 180,E1 -7472.59,E2 -7472.59} C_VEL
LIN {X 0,Y 466.774,Z 527.537,A -85,B 0,C 180,E1 -7473.453,E2 -7473.453} C_VEL
LIN {X 0,Y 466.745,Z 524.677,A -85,B 0,C 180,E1 -7474.751,E2 -7474.751} C_VEL
LIN {X 0,Y 466.993,Z 520.791,A -85,B 0,C 180,E1 -7476.047,E2 -7476.047} C_VEL
LIN {X 0,Y 467.099,Z 515.783,A -85,B 0,C 180,E1 -7477.348,E2 -7477.348} C_VEL
LIN {X 0,Y 467.406,Z 509.477,A -85,B 0,C 180,E1 -7478.648,E2 -7478.648} C_VEL
LIN {X 0,Y 467.738,Z 501.581,A -85,B 0,C 180,E1 -7479.95,E2 -7479.95} C_VEL
LIN {X 0,Y 468.139,Z 493.531,A -85,B 0,C 180,E1 -7481.035,E2 -7481.035} C_VEL
LIN {X 0,Y 468.704,Z 483.703,A -85,B 0,C 180,E1 -7482.118,E2 -7482.118} C_VEL
LIN {X 0,Y 469.164,Z 472.518,A -85,B 0,C 180,E1 -7483.106,E2 -7483.106} C_VEL
LIN {X 0,Y 469.624,Z 461.823,A -85,B 0,C 180,E1 -7483.854,E2 -7483.854} C_VEL
LIN {X 0,Y 470.061,Z 449.858,A -85,B 0,C 180,E1 -7484.503,E2 -7484.503} C_VEL
LIN {X 0,Y 469.993,Z 442.092,A -85,B 0,C 180,E1 -7484.841,E2 -7484.841} C_VEL
LIN {X 0,Y 467.404,Z 428.924,A -85,B 0,C 180,E1 -7485.339,E2 -7485.339} C_VEL
LIN {X 0,Y 466.888,Z 426.378,A -85,B 0,C 180,E1 -7485.436,E2 -7485.436} C_VEL
LIN {X 0,Y 466.916,Z 421.529,A -85,B 0,C 180,E1 -7488.508,E2 -7488.508} C_VEL
LIN {X 0,Y 466.949,Z 416.058,A -85,B 0,C 180,E1 -7492.103,E2 -7492.103} C_VEL
LIN {X 0,Y 467.087,Z 411.938,A -85,B 0,C 180,E1 -7494.917,E2 -7494.917} C_VEL
LIN {X 0,Y 467.182,Z 407.808,A -85,B 0,C 180,E1 -7497.797,E2 -7497.797} C_VEL
LIN {X 0,Y 467.358,Z 403.636,A -85,B 0,C 180,E1 -7500.749,E2 -7500.749} C_VEL
LIN {X 0,Y 467.465,Z 398.882,A -85,B 0,C 180,E1 -7504.219,E2 -7504.219} C_VEL
LIN {X 0,Y 467.455,Z 397.258,A -85,B 0,C 180,E1 -7505.721,E2 -7505.721} C_VEL
LIN {X 0,Y 467.563,Z 397.246,A -85,B 0,C 180,E1 -7508.591,E2 -7508.591} C_VEL
LIN {X 0,Y 467.584,Z 397.241,A -85,B 0,C 180,E1 -7511.402,E2 -7511.402} C_VEL
LIN {X 0,Y 467.567,Z 397.243,A -85,B 0,C 180,E1 -7513.822,E2 -7513.822} C_VEL
LIN {X 0,Y 467.554,Z 397.244,A -85,B 0,C 180,E1 -7516.255,E2 -7516.255} C_VEL
LIN {X 0,Y 467.581,Z 397.244,A -85,B 0,C 180,E1 -7518.723,E2 -7518.723} C_VEL
LIN {X 0,Y 467.568,Z 397.241,A -85,B 0,C 180,E1 -7521.956,E2 -7521.956} C_VEL
LIN {X 0,Y 467.567,Z 397.243,A -85,B 0,C 180,E1 -7525.167,E2 -7525.167} C_VEL
LIN {X 0,Y 467.586,Z 397.241,A -85,B 0,C 180,E1 -7528.26,E2 -7528.26} C_VEL
LIN {X 0,Y 467.58,Z 397.24,A -85,B 0,C 180,E1 -7531.25,E2 -7531.25} C_VEL
LIN {X 0,Y 467.616,Z 397.234,A -85,B 0,C 180,E1 -7533.199,E2 -7533.199} C_VEL
LIN {X 0,Y 467.594,Z 397.24,A -85,B 0,C 180,E1 -7536.469,E2 -7536.469} C_VEL
LIN {X 0,Y 467.627,Z 397.238,A -85,B 0,C 180,E1 -7539.777,E2 -7539.777} C_VEL
LIN {X 0,Y 467.602,Z 397.24,A -85,B 0,C 180,E1 -7542.506,E2 -7542.506} C_VEL
LIN {X 0,Y 467.61,Z 397.236,A -85,B 0,C 180,E1 -7545.196,E2 -7545.196} C_VEL
LIN {X 0,Y 467.66,Z 397.232,A -85,B 0,C 180,E1 -7547.855,E2 -7547.855} C_VEL
LIN {X 0,Y 467.685,Z 397.228,A -85,B 0,C 180,E1 -7551.357,E2 -7551.357} C_VEL
LIN {X 0,Y 467.747,Z 397.221,A -85,B 0,C 180,E1 -7553.963,E2 -7553.963} C_VEL
LIN {X 0,Y 467.861,Z 397.206,A -85,B 0,C 180,E1 -7557.417,E2 -7557.417} C_VEL
LIN {X 0,Y 467.885,Z 397.206,A -85,B 0,C 180,E1 -7560,E2 -7560} C_VEL
LIN {X 0,Y 467.862,Z 397.204,A -85,B 0,C 180,E1 -7562.583,E2 -7562.583} C_VEL
LIN {X 0,Y 467.747,Z 397.22,A -85,B 0,C 180,E1 -7566.037,E2 -7566.037} C_VEL
LIN {X 0,Y 467.685,Z 397.228,A -85,B 0,C 180,E1 -7568.643,E2 -7568.643} C_VEL
LIN {X 0,Y 467.687,Z 397.228,A -85,B 0,C 180,E1 -7572.145,E2 -7572.145} C_VEL
LIN {X 0,Y 467.653,Z 397.231,A -85,B 0,C 180,E1 -7575.885,E2 -7575.885} C_VEL
LIN {X 0,Y 467.628,Z 397.237,A -85,B 0,C 180,E1 -7579.308,E2 -7579.308} C_VEL
LIN {X 0,Y 467.537,Z 397.247,A -85,B 0,C 180,E1 -7582.074,E2 -7582.074} C_VEL
LIN {X 0,Y 467.588,Z 397.24,A -85,B 0,C 180,E1 -7584.888,E2 -7584.888} C_VEL
LIN {X 0,Y 467.63,Z 397.234,A -85,B 0,C 180,E1 -7587.768,E2 -7587.768} C_VEL
LIN {X 0,Y 467.571,Z 397.246,A -85,B 0,C 180,E1 -7591.045,E2 -7591.045} C_VEL
LIN {X 0,Y 467.592,Z 397.24,A -85,B 0,C 180,E1 -7594.242,E2 -7594.242} C_VEL
LIN {X 0,Y 467.553,Z 397.246,A -85,B 0,C 180,E1 -7597.187,E2 -7597.187} C_VEL
LIN {X 0,Y 467.58,Z 397.239,A -85,B 0,C 180,E1 -7600.264,E2 -7600.264} C_VEL
LIN {X 0,Y 467.589,Z 397.24,A -85,B 0,C 180,E1 -7602.567,E2 -7602.567} C_VEL
LIN {X 0,Y 467.573,Z 397.242,A -85,B 0,C 180,E1 -7605.053,E2 -7605.053} C_VEL
LIN {X 0,Y 467.591,Z 397.241,A -85,B 0,C 180,E1 -7607.44,E2 -7607.44} C_VEL
LIN {X 0,Y 467.632,Z 397.347,A -85,B 0,C 180,E1 -7611.024,E2 -7611.024} C_VEL
LIN {X 0,Y 468.452,Z 402.473,A -85,B 0,C 180,E1 -7613.653,E2 -7613.653} C_VEL
LIN {X 0,Y 468.491,Z 406.496,A -85,B 0,C 180,E1 -7615.596,E2 -7615.596} C_VEL
LIN {X 0,Y 468.228,Z 412.352,A -85,B 0,C 180,E1 -7618.309,E2 -7618.309} C_VEL
LIN {X 0,Y 468.041,Z 417.376,A -85,B 0,C 180,E1 -7620.566,E2 -7620.566} C_VEL
LIN {X 0,Y 467.651,Z 425.655,A -85,B 0,C 180,E1 -7624.162,E2 -7624.162} C_VEL
LIN {X 0,Y 467.404,Z 433.465,A -85,B 0,C 180,E1 -7627.454,E2 -7627.454} C_VEL
LIN {X 0,Y 467.216,Z 440.094,A -85,B 0,C 180,E1 -7630.217,E2 -7630.217} C_VEL
LIN {X 0,Y 467.041,Z 447.78,A -85,B 0,C 180,E1 -7633.387,E2 -7633.387} C_VEL
LIN {X 0,Y 466.982,Z 450.82,A -85,B 0,C 180,E1 -7634.603,E2 -7634.603} C_VEL
LIN {X 0,Y 469.081,Z 464.037,A -85,B 0,C 180,E1 -7635.024,E2 -7635.024} C_VEL
LIN {X 0,Y 470.026,Z 471.28,A -85,B 0,C 180,E1 -7635.33,E2 -7635.33} C_VEL
LIN {X 0,Y 469.593,Z 483.617,A -85,B 0,C 180,E1 -7635.924,E2 -7635.924} C_VEL
